// TwinCAT 3 PLC project Rohlik_Expansion
// ProgramVersion: 3.1.4024.0
// libraries:
//   CmpBitmapPool, * (System)
//   Tc2_EtherCAT, * (Beckhoff Automation GmbH)
//   Tc2_IoFunctions, * (Beckhoff Automation GmbH)
//   Tc2_MC2, * (Beckhoff Automation GmbH)
//   Tc2_ModbusSrv, * (Beckhoff Automation GmbH)
//   Tc2_Standard, * (Beckhoff Automation GmbH)
//   Tc2_SUPS, * (Beckhoff Automation GmbH)
//   Tc2_System, * (Beckhoff Automation GmbH)
//   Tc2_Utilities, * (Beckhoff Automation GmbH)
//   Tc3_Module, * (Beckhoff Automation GmbH)
//   Tc3_PackML_V2, * (Beckhoff Automation GmbH)
//   Util, * (System)
//   VisuDialogs, * (System)
// project tree:
//   02DUTs/ E_PMLUserUnitMode.TcDUT (not stored), E_UnitName.TcDUT (not stored), ModuleID.TcDUT (not stored), ST_ChangeIntoProduction.TcDUT (not stored), ST_UnitInfo.TcDUT (not stored)
//   Ads/ AbortToteRequestParams.TcDUT (not stored), AutostoreControlCommand.TcDUT (not stored), BarcodeValidationRequestParams.TcDUT (not stored), BarcodeVerificationResult.TcDUT (not stored), ButtonStatus.TcDUT (not stored), AirPressureStatus.TcDUT (not stored), DigitalInputStatus.TcDUT (not stored), DigitalOutputStatus.TcDUT (not stored), AutostoreStatus.TcDUT, EStopStatus.TcDUT (not stored), E_SAFETYDOOR.TcDUT (not stored), E_SafetyStates.TcDUT (not stored), FB_AirPressure_Subsystem.TcPOU, FB_HeartBeat_Subsystem.TcPOU, FB_Light_tower_module.TcPOU (not stored), FB_MachineControl_Subsystem.TcPOU (not stored), FB_Safety_Subsystem.TcPOU, FB_Tote_Subsystem.TcPOU, GeneralStatus.TcDUT (not stored), HeartbeatParams.TcDUT (not stored), InboundToteParams.TcDUT (not stored), InitToteRequestParams.TcDUT (not stored), LightCurtainStatus.TcDUT (not stored), MachineCommandStructure.TcDUT (not stored), MachineControlCommand.TcDUT (not stored), MachineControlCommand_1.TcDUT (not stored), MachineStatus.TcDUT (not stored), MethodCallReturnValue.TcDUT (not stored), ModelIdentifier.TcDUT (not stored), OrderToteCommand.TcDUT (not stored), OutboundToteParams.TcDUT (not stored), PerturbToteParams.TcDUT (not stored), SafetyDoorStatus.TcDUT (not stored), SafetyStatus.TcDUT (not stored), SensorStatus.TcDUT (not stored), StationMode.TcDUT (not stored), ST_BagOpen.TcDUT (not stored), ST_LightTower.TcDUT (not stored), SwapToteParams.TcDUT (not stored), ToteData.TcPOU (not stored), UpdateLightTowerParams.TcDUT (not stored), UpdateStationModeParams.TcDUT (not stored)
//   Ads/Ads/ BagOpeningStatus.TcPOU (not stored), ST_LightTowerAction.TcDUT (not stored)
//   GVLs/ GVL.TcGVL (not stored), GVL_SAFETY.TcGVL, G_HMI.TcGVL (not stored), G_IO.TcGVL (not stored), ST_Ifm_Qualifier.TcDUT (not stored), ST_Ifm_RX.TcDUT (not stored), ST_Ifm_TX.TcDUT (not stored), ST_IO_16.TcDUT (not stored), ST_SafetyIO.TcDUT (not stored)
//   / EtherCAT_Task.TcTTO (not stored), GlobalTextList.TcGTLO, MianTask.TcTTO (not stored), VisualizationManager.TcVMO (not stored), VISU_TASK.TcTTO (not stored)
//   LogTECH/ LogTechControlCmd.TcDUT (not stored), LogTechStatus.TcDUT (not stored), LogTechTransferStatus.TcDUT (not stored)
//   Mian/axis/ AxisHMI_Ex.TcVIS (not stored), E_HomingSteps.TcDUT (not stored), FB_MotionAxis_MC.TcPOU (not stored), MC_HomeAxis.TcPOU (not stored), ST_MotionAxis_MC.TcDUT (not stored)
//   Mian/DUTs/ BagStatus.TcDUT (not stored), Buffer_roller.TcDUT (not stored), E_Condition.TcDUT (not stored), E_LoadingStates.TcDUT (not stored), E_SampleStates.TcDUT (not stored), E_RollerStates.TcDUT (not stored), E_AutoStore_States.TcDUT (not stored), E_topic_sample.TcDUT (not stored), E_Transfer.TcDUT (not stored), E_WorkingStates.TcDUT, FB_DigitalInput.TcPOU (not stored), FB_GPWM.TcPOU (not stored), Inbound.TcDUT (not stored), I_Common.TcIO (not stored), OrderToteErrorStatus.TcDUT (not stored), Outbound.TcDUT (not stored), Prepare_Date_Time.TcPOU (not stored), Roller.TcDUT (not stored), Roller_x.TcDUT (not stored), Roller_y.TcDUT (not stored), ServerityLevelType.TcDUT (not stored), ST_Alarm_Hmi.TcDUT (not stored), ST_control_pannel.TcDUT (not stored), ST_EVENT.TcDUT (not stored), ST_safetyDoor.TcDUT (not stored), ToteStatus.TcDUT (not stored), ToteSubsystemWorkflowStatus.TcDUT (not stored), Valve.TcDUT (not stored)
//   Mian/ FB_Generic.TcPOU (not stored), FB_Machine.TcPOU (not stored), FB_mcp.TcPOU (not stored), FB_Sample.TcPOU (not stored), FB_loading_tote.TcPOU, FB_autoStore.TcPOU, FB_StateMachine.TcPOU, FB_working_tote.TcPOU, FB_Visu.TcPOU (not stored), FB_WriteLog.TcPOU (not stored), MAIN.TcPOU
//   PubSub/ E_Topics.TcDUT (not stored), I_PubSubService.TcIO (not stored), I_SubCallback.TcIO (not stored), KeyAndValue.TcDUT (not stored), PubSubData.TcDUT (not stored), PubSubService.TcPOU (not stored), ST_TracePublish.TcDUT (not stored), SubscriberCell.TcDUT (not stored)
//   VISUs/ ImagePool.TcIPO (not stored), visu_main.TcVIS (not stored)
//   VISUs/Templates/ visu_autoStore.TcVIS, VIS_TemplateCommand.TcVIS (not stored), VIS_TemplateKeys.TcVIS (not stored), VIS_TemplateMachine.TcVIS (not stored), VIS_TemplatePMLStateModel.TcVIS (not stored), VIS_TemplateToProduction.TcVIS (not stored), v_io_autoStore.TcVIS
//   VISUs/VISUs/ Menu.TcVIS, visu_2sys.TcVIS (not stored), visu_autoStore2.TcVIS, visu_loading.TcVIS (not stored), visu_operation.TcVIS, visu_sample.TcVIS (not stored), visu_manual.TcVIS, visu_working1.TcVIS (not stored), visu_autoStore1.TcVIS (not stored), visu_working2.TcVIS (not stored), v_alarm.TcVIS (not stored), v_io_loading.TcVIS (not stored), v_io_working1.TcVIS (not stored), v_io_working2.TcVIS
// real-time tasks:
//   TASK PlcTask: cycle T#4ms, priority 20, ADS port 350
//   TASK EtherCAT_Task: cycle T#2ms, priority 2, ADS port 351
//   TASK VISU_TASK: cycle T#100000us, priority 30, ADS port 352
// motion (NC):
//   TASK NC-Task 1 SAF: cycle T#2ms, priority 4, ADS port 501
//   TASK NC-Task 1 SVB: cycle T#10ms, priority 8, ADS port 511
//   AXIS lift_motor (id 3)
//     Velo: SlowManual=5, FastManual=20
//     PositionAreaControl: Enable=false
//     OtherSettings: AllowMotionCmdToSlave=true
//     encoder EncType=19
//       EncPara: ScaleFactorNumerator=3.333333333333, ScaleFactorDenominator=8388608, Inverse=true, MaxCount=#xffffffff, ReferenceSystem=1
//         SoftEndMinControl: Enable=true, Range=-5
//         SoftEndMaxControl: Enable=true, Range=800
//         Inc: RefSoftSyncMask=#x00800000
//     drive DrvType=16
//       DrvPara: Inverse=true, MaxCount=#xffffffff, DriveControlDWord=#x00020100
//         Analog: TorqueSetpointScale=10, ScaleFactorActTorque=0.1
//         TimeComp: TaskDelayCycles=1
//     controller CtrType=1
//       CtrPara: PriorControlFactor=1
//         PosDiffControl: Enable=false
//         Observer: BandWidth=20
//   AXIS working1_lift_motor (id 4)
//     PositionAreaControl: Enable=false
//     OtherSettings: AllowMotionCmdToSlave=true
//     encoder EncType=19
//       EncPara: ScaleFactorNumerator=5, ScaleFactorDenominator=8388608, Inverse=true, MaxCount=#xffffffff, ReferenceSystem=1
//         SoftEndMinControl: Enable=true, Range=-5
//         SoftEndMaxControl: Enable=true, Range=140
//         Inc: RefSoftSyncMask=#x00800000
//     drive DrvType=16
//       DrvPara: Inverse=true, MaxCount=#xffffffff, DriveControlDWord=#x00020100
//         Analog: TorqueSetpointScale=10, ScaleFactorActTorque=0.1
//         TimeComp: TaskDelayCycles=1
//     controller CtrType=1
//       CtrPara: PriorControlFactor=1
//         PosDiffControl: Enable=false
//         Observer: BandWidth=20
//   AXIS working1_open_bag (id 5)
//     General: UnitName=°
//     Dynamic: Acceleration=75, Deceleration=75, Jerk=112.5
//     Velo: SlowManual=1, FastManual=5, Maximum=300
//     PositionAreaControl: Enable=false
//     OtherSettings: AllowMotionCmdToSlave=true
//     encoder EncType=19
//       EncPara: ScaleFactorNumerator=36, ScaleFactorDenominator=8388608, MaxCount=#xffffffff, ReferenceSystem=1
//         SoftEndMinControl: Enable=true
//         SoftEndMaxControl: Enable=true, Range=60
//         Inc: RefSoftSyncMask=#x00800000
//     drive DrvType=16
//       DrvPara: MaxCount=#xffffffff, DriveControlDWord=#x00020100
//         Analog: TorqueSetpointScale=10, ScaleFactorActTorque=0.1
//         TimeComp: TaskDelayCycles=1
//     controller CtrType=1
//       CtrPara: PriorControlFactor=1
//         PosDiffControl: Enable=false
//         Observer: BandWidth=20
//   AXIS working2_lift_motor (id 1)
//     PositionAreaControl: Enable=false
//     OtherSettings: AllowMotionCmdToSlave=true
//     encoder EncType=19
//       EncPara: ScaleFactorNumerator=5, ScaleFactorDenominator=8388608, Inverse=true, MaxCount=#xffffffff, ReferenceSystem=1
//         SoftEndMinControl: Enable=true, Range=-5
//         SoftEndMaxControl: Enable=true, Range=140
//         Inc: RefSoftSyncMask=#x00800000
//     drive DrvType=16
//       DrvPara: Inverse=true, MaxCount=#xffffffff, DriveControlDWord=#x00020100
//         Analog: TorqueSetpointScale=10, ScaleFactorActTorque=0.1
//         TimeComp: TaskDelayCycles=1
//     controller CtrType=1
//       CtrPara: PriorControlFactor=1
//         PosDiffControl: Enable=false
//         Observer: BandWidth=20
//   AXIS working2_open_bag (id 2)
//     General: UnitName=°
//     Dynamic: Acceleration=75, Deceleration=75, Jerk=112.5
//     Velo: Maximum=300
//     PositionAreaControl: Enable=false
//     OtherSettings: AllowMotionCmdToSlave=true
//     encoder EncType=19
//       EncPara: ScaleFactorNumerator=36, ScaleFactorDenominator=8388608, MaxCount=#xffffffff, ReferenceSystem=1
//         SoftEndMinControl: Enable=true
//         SoftEndMaxControl: Enable=true, Range=60
//         Inc: RefSoftSyncMask=#x00800000
//     drive DrvType=16
//       DrvPara: MaxCount=#xffffffff, DriveControlDWord=#x00020100
//         Analog: TorqueSetpointScale=10, ScaleFactorActTorque=0.1
//         TimeComp: TaskDelayCycles=1
//     controller CtrType=1
//       CtrPara: PriorControlFactor=1
//         PosDiffControl: Enable=false
//         Observer: BandWidth=20
//   AXIS autostore1_transfer (id 12)
//     General: UnitName=°
//     Dynamic: Acceleration=75, Deceleration=75, Jerk=112.5
//     Velo: Maximum=600
//     PositionAreaControl: Enable=false
//     OtherSettings: AllowMotionCmdToSlave=true
//     encoder EncType=19
//       EncPara: ScaleFactorNumerator=34.6, ScaleFactorDenominator=8388608, Inverse=true, MaxCount=#xffffffff, ReferenceSystem=1
//         SoftEndMaxControl: Range=56
//         Inc: RefSoftSyncMask=#x00800000
//     drive DrvType=16
//       DrvPara: Inverse=true, MaxCount=#xffffffff, DriveControlDWord=#x00000100
//         Analog: TorqueSetpointScale=10, ScaleFactorActTorque=0.1
//         TimeComp: TaskDelayCycles=1
//     controller CtrType=1
//       CtrPara: PriorControlFactor=1
//         PosDiffControl: Enable=false
//         Observer: BandWidth=20
//   AXIS autostore1_lift (id 13)
//     General: UnitName=°
//     Dynamic: Acceleration=75, Deceleration=75, Jerk=112.5
//     Velo: Maximum=400
//     PositionAreaControl: Enable=false
//     OtherSettings: AllowMotionCmdToSlave=true
//     encoder EncType=19
//       EncPara: ScaleFactorNumerator=40, ScaleFactorDenominator=8388608, MaxCount=#xffffffff, ReferenceSystem=1
//         SoftEndMaxControl: Range=56
//         Inc: RefSoftSyncMask=#x00800000
//     drive DrvType=16
//       DrvPara: MaxCount=#xffffffff, DriveControlDWord=#x00000100
//         Analog: TorqueSetpointScale=10, ScaleFactorActTorque=0.1
//         TimeComp: TaskDelayCycles=1
//     controller CtrType=1
//       CtrPara: PriorControlFactor=1
//         PosDiffControl: Enable=false
//         Observer: BandWidth=20
//   AXIS autostore2_lift (id 7)
//     General: UnitName=°
//     Dynamic: Acceleration=75, Deceleration=75, Jerk=112.5
//     Velo: Maximum=400
//     PositionAreaControl: Enable=false
//     OtherSettings: AllowMotionCmdToSlave=true
//     encoder EncType=19
//       EncPara: ScaleFactorNumerator=40, ScaleFactorDenominator=8388608, MaxCount=#xffffffff, ReferenceSystem=1
//         SoftEndMaxControl: Range=56
//         Inc: RefSoftSyncMask=#x00800000
//     drive DrvType=16
//       DrvPara: MaxCount=#xffffffff, DriveControlDWord=#x00020100
//         Analog: TorqueSetpointScale=10, ScaleFactorActTorque=0.1
//         TimeComp: TaskDelayCycles=1
//     controller CtrType=1
//       CtrPara: PriorControlFactor=1
//         PosDiffControl: Enable=false
//         Observer: BandWidth=20
//   AXIS autostore2_transfer (id 6)
//     General: UnitName=°
//     Dynamic: Acceleration=75, Deceleration=75, Jerk=112.5
//     Velo: Maximum=600
//     PositionAreaControl: Enable=false
//     OtherSettings: AllowMotionCmdToSlave=true
//     encoder EncType=19
//       EncPara: ScaleFactorNumerator=34.6, ScaleFactorDenominator=8388608, Inverse=true, MaxCount=#xffffffff, ReferenceSystem=1
//         SoftEndMaxControl: Range=56
//         Inc: RefSoftSyncMask=#x00800000
//     drive DrvType=16
//       DrvPara: Inverse=true, MaxCount=#xffffffff, DriveControlDWord=#x00020100
//         Analog: TorqueSetpointScale=10, ScaleFactorActTorque=0.1
//         TimeComp: TaskDelayCycles=1
//     controller CtrType=1
//       CtrPara: PriorControlFactor=1
//         PosDiffControl: Enable=false
//         Observer: BandWidth=20
// I/O:
//   DEVICE Device 2 (RT-Ethernet Adapter)
//   DEVICE MCP, AmsNetId 192.168.17.27.4.1
//     Box 1 (CU2508) [CU2508 Ethernet Port]
//     MCP-EK1100 [EK1100 EtherCAT Coupler (2A E-Bus)]
//       DI0 [EL1809 16Ch. Dig. Input 24V, 3ms]
//       DI1 [EL1809 16Ch. Dig. Input 24V, 3ms]
//       DO0 [EL2809 16Ch. Dig. Output 24V, 0.5A]
//       DO1 [EL2809 16Ch. Dig. Output 24V, 0.5A]
//       Term 7 (EL6910) [EL6910, TwinSAFE PLC]
//       SI0 [EL1904, 4 Ch. Safety Input 24V, TwinSAFE]
//         modules: Module 1 (FSOES)
//       SI1 [EL1904, 4 Ch. Safety Input 24V, TwinSAFE]
//         modules: Module 1 (FSOES)
//       SI2 [EL1904, 4 Ch. Safety Input 24V, TwinSAFE]
//         modules: Module 1 (FSOES)
//       SI3 [EL1904, 4 Ch. Safety Input 24V, TwinSAFE]
//         modules: Module 1 (FSOES)
//       SO0 [EL2904, 4 Ch. Safety Output 24V, 0.5A, TwinSAFE]
//         modules: Module 1 (FSOES), Module 2 (DO)
//       SO4 [EL2904, 4 Ch. Safety Output 24V, 0.5A, TwinSAFE]
//         modules: Module 1 (FSOES), Module 2 (DO)
//       Term 50 (EL9410) [EL9410 E-Bus Power Supplier  (Diagnostics)]
//       Term 13 (EL3064) [EL3064 4Ch. Ana. Input 0-10V]
//       SI7 [EL1904, 4 Ch. Safety Input 24V, TwinSAFE]
//         modules: Module 1 (FSOES)
//       SI8 [EL1904, 4 Ch. Safety Input 24V, TwinSAFE]
//         modules: Module 1 (FSOES)
//       SO5 [EL2904, 4 Ch. Safety Output 24V, 0.5A, TwinSAFE]
//         modules: Module 1 (FSOES), Module 2 (DO)
//       SO6 [EL2904, 4 Ch. Safety Output 24V, 0.5A, TwinSAFE]
//         modules: Module 1 (FSOES), Module 2 (DO)
//       Term 14 (EL6631-0010) [EL6631-0010 PROFINET IO Device]
//       Term 15 (EL9011) [EL9011 End Terminal]
//   DEVICE Lift, AmsNetId 192.168.17.27.5.1
//     Box 16 (CU2508) [CU2508 Ethernet Port]
//     Term 17 (EK1100) [EK1100 EtherCAT Coupler (2A E-Bus)]
//       DI2 [EL1809 16Ch. Dig. Input 24V, 3ms]
//       DI3 [EL1809 16Ch. Dig. Input 24V, 3ms]
//       DO2 [EL2809 16Ch. Dig. Output 24V, 0.5A]
//       DO3 [EL2809 16Ch. Dig. Output 24V, 0.5A]
//       SI4 [EL1904, 4 Ch. Safety Input 24V, TwinSAFE]
//         modules: Module 1 (FSOES)
//       SI5 [EL1904, 4 Ch. Safety Input 24V, TwinSAFE]
//         modules: Module 1 (FSOES)
//       SI6 [EL1904, 4 Ch. Safety Input 24V, TwinSAFE]
//         modules: Module 1 (FSOES)
//       SO1 [EL2904, 4 Ch. Safety Output 24V, 0.5A, TwinSAFE]
//         modules: Module 1 (FSOES), Module 2 (DO)
//       Term 10 (EL9011) [EL9011 End Terminal]
//     lift_lift [SV660_1Axis_00915]
//     Box 26 (ifm IO-Link Master AL1332) [ifm IO-Link Master AL1332]
//       modules: Module 1 (IOL_4/4_I/O-Bytes), Module 2 (IOL_4/4_I/O-Bytes), Module 3 (IOL_4/4_I/O-Bytes), Module 4 (IOL_4/4_I/O-Bytes), Module 5 (IOL_4/4_I/O-Bytes), Module 6 (IOL_4/4_I/O-Bytes), Module 7 (IOL_4/4_I/O-Bytes), Module 8 (IOL_4/4_I/O-Bytes)
//   DEVICE Place1, AmsNetId 192.168.17.27.6.1
//     Box 26 (CU2508) [CU2508 Ethernet Port]
//     Term 27 (EK1100) [EK1100 EtherCAT Coupler (2A E-Bus)]
//       DI4 [EL1809 16Ch. Dig. Input 24V, 3ms]
//       DI5 [EL1809 16Ch. Dig. Input 24V, 3ms]
//       DO4 [EL2809 16Ch. Dig. Output 24V, 0.5A]
//       SO2 [EL2904, 4 Ch. Safety Output 24V, 0.5A, TwinSAFE]
//         modules: Module 1 (FSOES), Module 2 (DO)
//       Term 53 (EL9410) [EL9410 E-Bus Power Supplier  (Diagnostics)]
//       DO6 [EL2809 16Ch. Dig. Output 24V, 0.5A]
//       Term 9 (EL9011) [EL9011 End Terminal]
//     place1_lift [SV660_1Axis_00915]
//     place_openbag [SV660_1Axis_00915]
//     Box 36 (ifm IO-Link Master AL1332) [ifm IO-Link Master AL1332]
//       modules: Module 1 (IOL_4/4_I/O-Bytes), Module 2 (IOL_4/4_I/O-Bytes), Module 3 (IOL_4/4_I/O-Bytes), Module 4 (IOL_4/4_I/O-Bytes), Module 5 (IOL_4/4_I/O-Bytes), Module 6 (IOL_4/4_I/O-Bytes), Module 7 (IOL_4/4_I/O-Bytes), Module 8 (IOL_4/4_I/O-Bytes)
//   DEVICE Place2, AmsNetId 192.168.17.27.7.1
//     Box 35 (CU2508) [CU2508 Ethernet Port]
//     Term 36 (EK1100) [EK1100 EtherCAT Coupler (2A E-Bus)]
//       DI6 [EL1809 16Ch. Dig. Input 24V, 3ms]
//       DI7 [EL1809 16Ch. Dig. Input 24V, 3ms]
//       DO5 [EL2809 16Ch. Dig. Output 24V, 0.5A]
//       SO3 [EL2904, 4 Ch. Safety Output 24V, 0.5A, TwinSAFE]
//         modules: Module 1 (FSOES), Module 2 (DO)
//       Term 51 (EL9410) [EL9410 E-Bus Power Supplier  (Diagnostics)]
//       DO7 [EL2809 16Ch. Dig. Output 24V, 0.5A]
//       Term 9 (EL9011) [EL9011 End Terminal]
//     place2_lift [SV660_1Axis_00915]
//     place2_openbag [SV660_1Axis_00915]
//     Box 46 (ifm IO-Link Master AL1332) [ifm IO-Link Master AL1332]
//       modules: Module 1 (IOL_4/4_I/O-Bytes), Module 2 (IOL_4/4_I/O-Bytes), Module 3 (IOL_4/4_I/O-Bytes), Module 4 (IOL_4/4_I/O-Bytes), Module 5 (IOL_4/4_I/O-Bytes), Module 6 (IOL_4/4_I/O-Bytes), Module 7 (IOL_4/4_I/O-Bytes), Module 8 (IOL_4/4_I/O-Bytes)
//   DEVICE Device 1 (EtherCAT Automation Protocol), AmsNetId 192.168.11.159.2.1
//   DEVICE autoStore1, AmsNetId 192.168.11.159.8.1
//     Box 55 (CU2508) [CU2508 Ethernet Port]
//     Term 56 (EK1100) [EK1100 EtherCAT Coupler (2A E-Bus)]
//       DI20 [EL1809 16Ch. Dig. Input 24V, 3ms]
//       Term 6 (EL9011) [EL9011 End Terminal]
//     autostore1_transfer [SV660_1Axis_00916]
//     autostore1_lift [SV660_1Axis_00916]
//   DEVICE autoStore2, AmsNetId 192.168.11.159.10.1
//     Box 65 (CU2508) [CU2508 Ethernet Port]
//     Term 70 (EK1100) [EK1100 EtherCAT Coupler (2A E-Bus)]
//       DI21 [EL1809 16Ch. Dig. Input 24V, 3ms]
//       Term 10 (EL9011) [EL9011 End Terminal]
//     autostore2_transfer [SV660_1Axis_00916]
//     autostore2_lift [SV660_1Axis_00916]
// variable links:
//   Lift <-> MCP/MCP-EK1100/Term 7 (EL6910)
//     Term 17 (EK1100)/SI5/Module 1 (FSOES)/RxPDO/FSOE <-> ConnectionInputs/Message_29 TxPDO
//     Term 17 (EK1100)/SI6/Module 1 (FSOES)/RxPDO/FSOE <-> ConnectionInputs/Message_30 TxPDO
//     Term 17 (EK1100)/SO1/Module 1 (FSOES)/TxPDO/FSOE <-> ConnectionOutputs/Message_31 RxPDO
//   MCP <-> Lift/Term 17 (EK1100)/SI4
//     MCP-EK1100/Term 7 (EL6910)/ConnectionInputs/Message_28 TxPDO <-> Module 1 (FSOES)/RxPDO/FSOE
//     MCP-EK1100/Term 7 (EL6910)/ConnectionOutputs/Message_28 RxPDO <-> Module 1 (FSOES)/TxPDO/FSOE
//   MCP <-> Lift/Term 17 (EK1100)/SI5
//     MCP-EK1100/Term 7 (EL6910)/ConnectionOutputs/Message_29 RxPDO <-> Module 1 (FSOES)/TxPDO/FSOE
//   MCP <-> Lift/Term 17 (EK1100)/SI6
//     MCP-EK1100/Term 7 (EL6910)/ConnectionOutputs/Message_30 RxPDO <-> Module 1 (FSOES)/TxPDO/FSOE
//   MCP <-> Lift/Term 17 (EK1100)/SO1
//     MCP-EK1100/Term 7 (EL6910)/ConnectionInputs/Message_31 TxPDO <-> Module 1 (FSOES)/RxPDO/FSOE
//   MCP <-> MCP/MCP-EK1100/SI0
//     MCP-EK1100/Term 7 (EL6910)/ConnectionInputs/Message_22 TxPDO <-> Module 1 (FSOES)/RxPDO/FSOE
//     MCP-EK1100/Term 7 (EL6910)/ConnectionOutputs/Message_22 RxPDO <-> Module 1 (FSOES)/TxPDO/FSOE
//   MCP <-> MCP/MCP-EK1100/SI1
//     MCP-EK1100/Term 7 (EL6910)/ConnectionInputs/Message_23 TxPDO <-> Module 1 (FSOES)/RxPDO/FSOE
//   MCP <-> MCP/MCP-EK1100/SI2
//     MCP-EK1100/Term 7 (EL6910)/ConnectionOutputs/Message_24 RxPDO <-> Module 1 (FSOES)/TxPDO/FSOE
//   MCP <-> MCP/MCP-EK1100/SI3
//     MCP-EK1100/Term 7 (EL6910)/ConnectionInputs/Message_27 TxPDO <-> Module 1 (FSOES)/RxPDO/FSOE
//   MCP <-> MCP/MCP-EK1100/SO0
//     MCP-EK1100/Term 7 (EL6910)/ConnectionInputs/Message_26 TxPDO <-> Module 1 (FSOES)/RxPDO/FSOE
//   MCP <-> MCP/MCP-EK1100/SO5
//     MCP-EK1100/Term 7 (EL6910)/ConnectionOutputs/Message_71 RxPDO <-> Module 1 (FSOES)/TxPDO/FSOE
//   MCP <-> MCP/MCP-EK1100/SO6
//     MCP-EK1100/Term 7 (EL6910)/ConnectionInputs/Message_72 TxPDO <-> Module 1 (FSOES)/RxPDO/FSOE
//   MCP <-> MCP/MCP-EK1100/Term 7 (EL6910)
//     MCP-EK1100/SI1/Module 1 (FSOES)/TxPDO/FSOE <-> ConnectionOutputs/Message_23 RxPDO
//     MCP-EK1100/SI3/Module 1 (FSOES)/TxPDO/FSOE <-> ConnectionOutputs/Message_27 RxPDO
//     MCP-EK1100/SI2/Module 1 (FSOES)/RxPDO/FSOE <-> ConnectionInputs/Message_24 TxPDO
//     MCP-EK1100/SO0/Module 1 (FSOES)/TxPDO/FSOE <-> ConnectionOutputs/Message_26 RxPDO
//     MCP-EK1100/SO4/Module 1 (FSOES)/TxPDO/FSOE <-> ConnectionOutputs/Message_36 RxPDO
//     MCP-EK1100/SO6/Module 1 (FSOES)/TxPDO/FSOE <-> ConnectionOutputs/Message_72 RxPDO
//     MCP-EK1100/SO4/Module 1 (FSOES)/RxPDO/FSOE <-> ConnectionInputs/Message_36 TxPDO
//     MCP-EK1100/SO5/Module 1 (FSOES)/RxPDO/FSOE <-> ConnectionInputs/Message_71 TxPDO
//   MCP <-> Place2/Term 36 (EK1100)/SO3
//     MCP-EK1100/Term 7 (EL6910)/ConnectionInputs/Message_33 TxPDO <-> Module 1 (FSOES)/RxPDO/FSOE
//     MCP-EK1100/Term 7 (EL6910)/ConnectionOutputs/Message_33 RxPDO <-> Module 1 (FSOES)/TxPDO/FSOE
//   Place1 <-> MCP/MCP-EK1100/Term 7 (EL6910)
//     Term 27 (EK1100)/SO2/Module 1 (FSOES)/RxPDO/FSOE <-> ConnectionInputs/Message_32 TxPDO
//     Term 27 (EK1100)/SO2/Module 1 (FSOES)/TxPDO/FSOE <-> ConnectionOutputs/Message_32 RxPDO
//   NC-Task 1 SAF/Axes/autostore1_lift <-> autoStore1/autostore1_lift
//     Drive/Inputs/In/nDataIn1 <-> Inputs/Following error actual value
//     Drive/Inputs/In/nDataIn3[0] <-> Inputs/Torque actual value
//     Drive/Inputs/In/nDcOutputTime <-> InfoData/DcOutputShift
//     Drive/Inputs/In/nState1 <-> Inputs/Statusword
//     Drive/Inputs/In/nState2 <-> Inputs/Statusword @bit 8
//     Drive/Inputs/In/nState4 @bit 1 <-> WcState/InputToggle
//     Drive/Inputs/In/nState4 <-> WcState/WcState
//     Drive/Outputs/Out/nCtrl1 <-> Outputs/Controlword
//     Drive/Outputs/Out/nCtrl2 <-> Outputs/Controlword @bit 8
//     Drive/Outputs/Out/nDataOut1 <-> Outputs/Target position
//     Enc/Inputs/In/nDataIn1 <-> Inputs/Position actual value
//     Enc/Inputs/In/nDataIn3 <-> Inputs/Touch probe pos1 pos value
//     Enc/Inputs/In/nDataIn5 <-> Inputs/Touch probe pos2 pos value
//     Enc/Inputs/In/nDcInputTime <-> InfoData/DcInputShift
//     Enc/Inputs/In/nState4 @bit 1 <-> WcState/InputToggle
//     Enc/Inputs/In/nState4 <-> WcState/WcState
//     Enc/Inputs/In/nState5 <-> Inputs/Touch probe status
//     Enc/Inputs/In/nState6 <-> Inputs/Touch probe status @bit 8
//     Enc/Outputs/Out/nCtrl5 <-> Outputs/Touch probe function
//     Enc/Outputs/Out/nCtrl6 <-> Outputs/Touch probe function @bit 8
//   NC-Task 1 SAF/Axes/autostore1_transfer <-> autoStore1/autostore1_transfer
//     Drive/Inputs/In/nDataIn1 <-> Inputs/Following error actual value
//     Drive/Inputs/In/nDataIn3[0] <-> Inputs/Torque actual value
//     Drive/Inputs/In/nDcOutputTime <-> InfoData/DcOutputShift
//     Drive/Inputs/In/nState1 <-> Inputs/Statusword
//     Drive/Inputs/In/nState2 <-> Inputs/Statusword @bit 8
//     Drive/Inputs/In/nState4 @bit 1 <-> WcState/InputToggle
//     Drive/Inputs/In/nState4 <-> WcState/WcState
//     Drive/Outputs/Out/nCtrl1 <-> Outputs/Controlword
//     Drive/Outputs/Out/nCtrl2 <-> Outputs/Controlword @bit 8
//     Drive/Outputs/Out/nDataOut1 <-> Outputs/Target position
//     Enc/Inputs/In/nDataIn1 <-> Inputs/Position actual value
//     Enc/Inputs/In/nDataIn3 <-> Inputs/Touch probe pos1 pos value
//     Enc/Inputs/In/nDataIn5 <-> Inputs/Touch probe pos2 pos value
//     Enc/Inputs/In/nDcInputTime <-> InfoData/DcInputShift
//     Enc/Inputs/In/nState4 @bit 1 <-> WcState/InputToggle
//     Enc/Inputs/In/nState4 <-> WcState/WcState
//     Enc/Inputs/In/nState5 <-> Inputs/Touch probe status
//     Enc/Inputs/In/nState6 <-> Inputs/Touch probe status @bit 8
//     Enc/Outputs/Out/nCtrl5 <-> Outputs/Touch probe function
//     Enc/Outputs/Out/nCtrl6 <-> Outputs/Touch probe function @bit 8
//   NC-Task 1 SAF/Axes/autostore2_lift <-> autoStore2/autostore2_lift
//     Drive/Inputs/In/nDataIn1 <-> Inputs/Following error actual value
//     Drive/Inputs/In/nDataIn3[0] <-> Inputs/Torque actual value
//     Drive/Inputs/In/nDcOutputTime <-> InfoData/DcOutputShift
//     Drive/Inputs/In/nState1 <-> Inputs/Statusword
//     Drive/Inputs/In/nState2 <-> Inputs/Statusword @bit 8
//     Drive/Inputs/In/nState4 @bit 1 <-> WcState/InputToggle
//     Drive/Inputs/In/nState4 <-> WcState/WcState
//     Drive/Outputs/Out/nCtrl1 <-> Outputs/Controlword
//     Drive/Outputs/Out/nCtrl2 <-> Outputs/Controlword @bit 8
//     Drive/Outputs/Out/nDataOut1 <-> Outputs/Target position
//     Enc/Inputs/In/nDataIn1 <-> Inputs/Position actual value
//     Enc/Inputs/In/nDataIn3 <-> Inputs/Touch probe pos1 pos value
//     Enc/Inputs/In/nDataIn5 <-> Inputs/Touch probe pos2 pos value
//     Enc/Inputs/In/nDcInputTime <-> InfoData/DcInputShift
//     Enc/Inputs/In/nState4 @bit 1 <-> WcState/InputToggle
//     Enc/Inputs/In/nState4 <-> WcState/WcState
//     Enc/Inputs/In/nState5 <-> Inputs/Touch probe status
//     Enc/Inputs/In/nState6 <-> Inputs/Touch probe status @bit 8
//     Enc/Outputs/Out/nCtrl5 <-> Outputs/Touch probe function
//     Enc/Outputs/Out/nCtrl6 <-> Outputs/Touch probe function @bit 8
//   NC-Task 1 SAF/Axes/autostore2_transfer <-> autoStore2/autostore2_transfer
//     Drive/Inputs/In/nDataIn1 <-> Inputs/Following error actual value
//     Drive/Inputs/In/nDataIn3[0] <-> Inputs/Torque actual value
//     Drive/Inputs/In/nDcOutputTime <-> InfoData/DcOutputShift
//     Drive/Inputs/In/nState1 <-> Inputs/Statusword
//     Drive/Inputs/In/nState2 <-> Inputs/Statusword @bit 8
//     Drive/Inputs/In/nState4 @bit 1 <-> WcState/InputToggle
//     Drive/Inputs/In/nState4 <-> WcState/WcState
//     Drive/Outputs/Out/nCtrl1 <-> Outputs/Controlword
//     Drive/Outputs/Out/nCtrl2 <-> Outputs/Controlword @bit 8
//     Drive/Outputs/Out/nDataOut1 <-> Outputs/Target position
//     Enc/Inputs/In/nDataIn1 <-> Inputs/Position actual value
//     Enc/Inputs/In/nDataIn3 <-> Inputs/Touch probe pos1 pos value
//     Enc/Inputs/In/nDataIn5 <-> Inputs/Touch probe pos2 pos value
//     Enc/Inputs/In/nDcInputTime <-> InfoData/DcInputShift
//     Enc/Inputs/In/nState4 @bit 1 <-> WcState/InputToggle
//     Enc/Inputs/In/nState4 <-> WcState/WcState
//     Enc/Inputs/In/nState5 <-> Inputs/Touch probe status
//     Enc/Inputs/In/nState6 <-> Inputs/Touch probe status @bit 8
//     Enc/Outputs/Out/nCtrl5 <-> Outputs/Touch probe function
//     Enc/Outputs/Out/nCtrl6 <-> Outputs/Touch probe function @bit 8
//   NC-Task 1 SAF/Axes/lift_motor <-> Lift/lift_lift
//     Drive/Inputs/In/nDataIn1 <-> Inputs/Following error actual value
//     Drive/Inputs/In/nDataIn3[0] <-> Inputs/Torque actual value
//     Drive/Inputs/In/nDcOutputTime <-> InfoData/DcOutputShift
//     Drive/Inputs/In/nState1 <-> Inputs/Statusword
//     Drive/Inputs/In/nState2 <-> Inputs/Statusword @bit 8
//     Drive/Inputs/In/nState4 @bit 1 <-> WcState/InputToggle
//     Drive/Inputs/In/nState4 <-> WcState/WcState
//     Drive/Outputs/Out/nCtrl1 <-> Outputs/Controlword
//     Drive/Outputs/Out/nCtrl2 <-> Outputs/Controlword @bit 8
//     Drive/Outputs/Out/nDataOut1 <-> Outputs/Target position
//     Enc/Inputs/In/nDataIn1 <-> Inputs/Position actual value
//     Enc/Inputs/In/nDataIn3 <-> Inputs/Touch probe pos1 pos value
//     Enc/Inputs/In/nDataIn5 <-> Inputs/Touch probe pos2 pos value
//     Enc/Inputs/In/nDcInputTime <-> InfoData/DcInputShift
//     Enc/Inputs/In/nState4 @bit 1 <-> WcState/InputToggle
//     Enc/Inputs/In/nState4 <-> WcState/WcState
//     Enc/Inputs/In/nState5 <-> Inputs/Touch probe status
//     Enc/Inputs/In/nState6 <-> Inputs/Touch probe status @bit 8
//     Enc/Outputs/Out/nCtrl5 <-> Outputs/Touch probe function
//     Enc/Outputs/Out/nCtrl6 <-> Outputs/Touch probe function @bit 8
//   NC-Task 1 SAF/Axes/working1_lift_motor <-> Place1/place1_lift
//     Drive/Inputs/In/nDataIn1 <-> Inputs/Following error actual value
//     Drive/Inputs/In/nDataIn3[0] <-> Inputs/Torque actual value
//     Drive/Inputs/In/nDcOutputTime <-> InfoData/DcOutputShift
//     Drive/Inputs/In/nState1 <-> Inputs/Statusword
//     Drive/Inputs/In/nState2 <-> Inputs/Statusword @bit 8
//     Drive/Inputs/In/nState4 @bit 1 <-> WcState/InputToggle
//     Drive/Inputs/In/nState4 <-> WcState/WcState
//     Drive/Outputs/Out/nCtrl1 <-> Outputs/Controlword
//     Drive/Outputs/Out/nCtrl2 <-> Outputs/Controlword @bit 8
//     Drive/Outputs/Out/nDataOut1 <-> Outputs/Target position
//     Enc/Inputs/In/nDataIn1 <-> Inputs/Position actual value
//     Enc/Inputs/In/nDataIn3 <-> Inputs/Touch probe pos1 pos value
//     Enc/Inputs/In/nDataIn5 <-> Inputs/Touch probe pos2 pos value
//     Enc/Inputs/In/nDcInputTime <-> InfoData/DcInputShift
//     Enc/Inputs/In/nState4 @bit 1 <-> WcState/InputToggle
//     Enc/Inputs/In/nState4 <-> WcState/WcState
//     Enc/Inputs/In/nState5 <-> Inputs/Touch probe status
//     Enc/Inputs/In/nState6 <-> Inputs/Touch probe status @bit 8
//     Enc/Outputs/Out/nCtrl5 <-> Outputs/Touch probe function
//     Enc/Outputs/Out/nCtrl6 <-> Outputs/Touch probe function @bit 8
//   NC-Task 1 SAF/Axes/working1_open_bag <-> Place1/place_openbag
//     Drive/Inputs/In/nDataIn1 <-> Inputs/Following error actual value
//     Drive/Inputs/In/nDataIn3[0] <-> Inputs/Torque actual value
//     Drive/Inputs/In/nDcOutputTime <-> InfoData/DcOutputShift
//     Drive/Inputs/In/nState1 <-> Inputs/Statusword
//     Drive/Inputs/In/nState2 <-> Inputs/Statusword @bit 8
//     Drive/Inputs/In/nState4 @bit 1 <-> WcState/InputToggle
//     Drive/Inputs/In/nState4 <-> WcState/WcState
//     Drive/Outputs/Out/nCtrl1 <-> Outputs/Controlword
//     Drive/Outputs/Out/nCtrl2 <-> Outputs/Controlword @bit 8
//     Drive/Outputs/Out/nDataOut1 <-> Outputs/Target position
//     Enc/Inputs/In/nDataIn1 <-> Inputs/Position actual value
//     Enc/Inputs/In/nDataIn3 <-> Inputs/Touch probe pos1 pos value
//     Enc/Inputs/In/nDataIn5 <-> Inputs/Touch probe pos2 pos value
//     Enc/Inputs/In/nDcInputTime <-> InfoData/DcInputShift
//     Enc/Inputs/In/nState4 @bit 1 <-> WcState/InputToggle
//     Enc/Inputs/In/nState4 <-> WcState/WcState
//     Enc/Inputs/In/nState5 <-> Inputs/Touch probe status
//     Enc/Inputs/In/nState6 <-> Inputs/Touch probe status @bit 8
//     Enc/Outputs/Out/nCtrl5 <-> Outputs/Touch probe function
//     Enc/Outputs/Out/nCtrl6 <-> Outputs/Touch probe function @bit 8
//   NC-Task 1 SAF/Axes/working2_lift_motor <-> Place2/place2_lift
//     Drive/Inputs/In/nDataIn1 <-> Inputs/Following error actual value
//     Drive/Inputs/In/nDataIn3[0] <-> Inputs/Torque actual value
//     Drive/Inputs/In/nDcOutputTime <-> InfoData/DcOutputShift
//     Drive/Inputs/In/nState1 <-> Inputs/Statusword
//     Drive/Inputs/In/nState2 <-> Inputs/Statusword @bit 8
//     Drive/Inputs/In/nState4 @bit 1 <-> WcState/InputToggle
//     Drive/Inputs/In/nState4 <-> WcState/WcState
//     Drive/Outputs/Out/nCtrl1 <-> Outputs/Controlword
//     Drive/Outputs/Out/nCtrl2 <-> Outputs/Controlword @bit 8
//     Drive/Outputs/Out/nDataOut1 <-> Outputs/Target position
//     Enc/Inputs/In/nDataIn1 <-> Inputs/Position actual value
//     Enc/Inputs/In/nDataIn3 <-> Inputs/Touch probe pos1 pos value
//     Enc/Inputs/In/nDataIn5 <-> Inputs/Touch probe pos2 pos value
//     Enc/Inputs/In/nDcInputTime <-> InfoData/DcInputShift
//     Enc/Inputs/In/nState4 @bit 1 <-> WcState/InputToggle
//     Enc/Inputs/In/nState4 <-> WcState/WcState
//     Enc/Inputs/In/nState5 <-> Inputs/Touch probe status
//     Enc/Inputs/In/nState6 <-> Inputs/Touch probe status @bit 8
//     Enc/Outputs/Out/nCtrl5 <-> Outputs/Touch probe function
//     Enc/Outputs/Out/nCtrl6 <-> Outputs/Touch probe function @bit 8
//   NC-Task 1 SAF/Axes/working2_open_bag <-> Place2/place2_openbag
//     Drive/Inputs/In/nDataIn1 <-> Inputs/Following error actual value
//     Drive/Inputs/In/nDataIn3[0] <-> Inputs/Torque actual value
//     Drive/Inputs/In/nDcOutputTime <-> InfoData/DcOutputShift
//     Drive/Inputs/In/nState1 <-> Inputs/Statusword
//     Drive/Inputs/In/nState2 <-> Inputs/Statusword @bit 8
//     Drive/Inputs/In/nState4 @bit 1 <-> WcState/InputToggle
//     Drive/Inputs/In/nState4 <-> WcState/WcState
//     Drive/Outputs/Out/nCtrl1 <-> Outputs/Controlword
//     Drive/Outputs/Out/nCtrl2 <-> Outputs/Controlword @bit 8
//     Drive/Outputs/Out/nDataOut1 <-> Outputs/Target position
//     Enc/Inputs/In/nDataIn1 <-> Inputs/Position actual value
//     Enc/Inputs/In/nDataIn3 <-> Inputs/Touch probe pos1 pos value
//     Enc/Inputs/In/nDataIn5 <-> Inputs/Touch probe pos2 pos value
//     Enc/Inputs/In/nDcInputTime <-> InfoData/DcInputShift
//     Enc/Inputs/In/nState4 @bit 1 <-> WcState/InputToggle
//     Enc/Inputs/In/nState4 <-> WcState/WcState
//     Enc/Inputs/In/nState5 <-> Inputs/Touch probe status
//     Enc/Inputs/In/nState6 <-> Inputs/Touch probe status @bit 8
//     Enc/Outputs/Out/nCtrl5 <-> Outputs/Touch probe function
//     Enc/Outputs/Out/nCtrl6 <-> Outputs/Touch probe function @bit 8
//   Rohlik_Expansion/Rohlik_Expansion Instance <-> Device 1 (EtherCAT Automation Protocol)
//     MianTask Inputs/G_IO.devState_Device1 <-> Inputs/DevState
//   Rohlik_Expansion/Rohlik_Expansion Instance <-> Lift
//     MianTask Inputs/G_IO.wcState_lift <-> Inputs/Frm0WcState
//   Rohlik_Expansion/Rohlik_Expansion Instance <-> Lift/Box 26 (ifm IO-Link Master AL1332)
//     MianTask Inputs/G_IO.arIOLinkQualifier_Lift/CH[{0..7}] <-> TxPDO IO-Link Port Qualifier/Qualifier of IO-Link Ch.{1..8}  (8 links)
//     MianTask Inputs/G_IO.arIOLinkTx_Lift[0]/InputByte[0] <-> Module 1 (IOL_4/4_I/O-Bytes)/TxPDO/input byte 0
//     MianTask Inputs/G_IO.arIOLinkTx_Lift[0]/InputByte[1] <-> Module 1 (IOL_4/4_I/O-Bytes)/TxPDO/input byte 1
//     MianTask Inputs/G_IO.arIOLinkTx_Lift[0]/InputByte[2] <-> Module 1 (IOL_4/4_I/O-Bytes)/TxPDO/input byte 2
//     MianTask Inputs/G_IO.arIOLinkTx_Lift[0]/InputByte[3] <-> Module 1 (IOL_4/4_I/O-Bytes)/TxPDO/input byte 3
//     MianTask Inputs/G_IO.arIOLinkTx_Lift[1]/InputByte[0] <-> Module 2 (IOL_4/4_I/O-Bytes)/TxPDO/input byte 0
//     MianTask Inputs/G_IO.arIOLinkTx_Lift[1]/InputByte[1] <-> Module 2 (IOL_4/4_I/O-Bytes)/TxPDO/input byte 1
//     MianTask Inputs/G_IO.arIOLinkTx_Lift[1]/InputByte[2] <-> Module 2 (IOL_4/4_I/O-Bytes)/TxPDO/input byte 2
//     MianTask Inputs/G_IO.arIOLinkTx_Lift[1]/InputByte[3] <-> Module 2 (IOL_4/4_I/O-Bytes)/TxPDO/input byte 3
//     MianTask Inputs/G_IO.arIOLinkTx_Lift[2]/InputByte[0] <-> Module 3 (IOL_4/4_I/O-Bytes)/TxPDO/input byte 0
//     MianTask Inputs/G_IO.arIOLinkTx_Lift[2]/InputByte[1] <-> Module 3 (IOL_4/4_I/O-Bytes)/TxPDO/input byte 1
//     MianTask Inputs/G_IO.arIOLinkTx_Lift[2]/InputByte[2] <-> Module 3 (IOL_4/4_I/O-Bytes)/TxPDO/input byte 2
//     MianTask Inputs/G_IO.arIOLinkTx_Lift[2]/InputByte[3] <-> Module 3 (IOL_4/4_I/O-Bytes)/TxPDO/input byte 3
//     MianTask Inputs/G_IO.arIOLinkTx_Lift[3]/InputByte[0] <-> Module 4 (IOL_4/4_I/O-Bytes)/TxPDO/input byte 0
//     MianTask Inputs/G_IO.arIOLinkTx_Lift[3]/InputByte[1] <-> Module 4 (IOL_4/4_I/O-Bytes)/TxPDO/input byte 1
//     MianTask Inputs/G_IO.arIOLinkTx_Lift[3]/InputByte[2] <-> Module 4 (IOL_4/4_I/O-Bytes)/TxPDO/input byte 2
//     MianTask Inputs/G_IO.arIOLinkTx_Lift[3]/InputByte[3] <-> Module 4 (IOL_4/4_I/O-Bytes)/TxPDO/input byte 3
//     MianTask Inputs/G_IO.arIOLinkTx_Lift[4]/InputByte[0] <-> Module 5 (IOL_4/4_I/O-Bytes)/TxPDO/input byte 0
//     MianTask Inputs/G_IO.arIOLinkTx_Lift[4]/InputByte[1] <-> Module 5 (IOL_4/4_I/O-Bytes)/TxPDO/input byte 1
//     MianTask Inputs/G_IO.arIOLinkTx_Lift[4]/InputByte[2] <-> Module 5 (IOL_4/4_I/O-Bytes)/TxPDO/input byte 2
//     MianTask Inputs/G_IO.arIOLinkTx_Lift[4]/InputByte[3] <-> Module 5 (IOL_4/4_I/O-Bytes)/TxPDO/input byte 3
//     MianTask Inputs/G_IO.arIOLinkTx_Lift[5]/InputByte[0] <-> Module 6 (IOL_4/4_I/O-Bytes)/TxPDO/input byte 0
//     MianTask Inputs/G_IO.arIOLinkTx_Lift[5]/InputByte[1] <-> Module 6 (IOL_4/4_I/O-Bytes)/TxPDO/input byte 1
//     MianTask Inputs/G_IO.arIOLinkTx_Lift[5]/InputByte[2] <-> Module 6 (IOL_4/4_I/O-Bytes)/TxPDO/input byte 2
//     MianTask Inputs/G_IO.arIOLinkTx_Lift[5]/InputByte[3] <-> Module 6 (IOL_4/4_I/O-Bytes)/TxPDO/input byte 3
//     MianTask Inputs/G_IO.arIOLinkTx_Lift[6]/InputByte[0] <-> Module 7 (IOL_4/4_I/O-Bytes)/TxPDO/input byte 0
//     MianTask Inputs/G_IO.arIOLinkTx_Lift[6]/InputByte[1] <-> Module 7 (IOL_4/4_I/O-Bytes)/TxPDO/input byte 1
//     MianTask Inputs/G_IO.arIOLinkTx_Lift[6]/InputByte[2] <-> Module 7 (IOL_4/4_I/O-Bytes)/TxPDO/input byte 2
//     MianTask Inputs/G_IO.arIOLinkTx_Lift[6]/InputByte[3] <-> Module 7 (IOL_4/4_I/O-Bytes)/TxPDO/input byte 3
//     MianTask Inputs/G_IO.arIOLinkTx_Lift[7]/InputByte[0] <-> Module 8 (IOL_4/4_I/O-Bytes)/TxPDO/input byte 0
//     MianTask Inputs/G_IO.arIOLinkTx_Lift[7]/InputByte[1] <-> Module 8 (IOL_4/4_I/O-Bytes)/TxPDO/input byte 1
//     MianTask Inputs/G_IO.arIOLinkTx_Lift[7]/InputByte[2] <-> Module 8 (IOL_4/4_I/O-Bytes)/TxPDO/input byte 2
//     MianTask Inputs/G_IO.arIOLinkTx_Lift[7]/InputByte[3] <-> Module 8 (IOL_4/4_I/O-Bytes)/TxPDO/input byte 3
//     MianTask Outputs/G_IO.arIOLinkRx_Lift[0]/OutputByte[0] <-> Module 1 (IOL_4/4_I/O-Bytes)/RxPDO/output byte 0
//     MianTask Outputs/G_IO.arIOLinkRx_Lift[0]/OutputByte[1] <-> Module 1 (IOL_4/4_I/O-Bytes)/RxPDO/output byte 1
//     MianTask Outputs/G_IO.arIOLinkRx_Lift[0]/OutputByte[2] <-> Module 1 (IOL_4/4_I/O-Bytes)/RxPDO/output byte 2
//     MianTask Outputs/G_IO.arIOLinkRx_Lift[0]/OutputByte[3] <-> Module 1 (IOL_4/4_I/O-Bytes)/RxPDO/output byte 3
//     MianTask Outputs/G_IO.arIOLinkRx_Lift[1]/OutputByte[0] <-> Module 2 (IOL_4/4_I/O-Bytes)/RxPDO/output byte 0
//     MianTask Outputs/G_IO.arIOLinkRx_Lift[1]/OutputByte[1] <-> Module 2 (IOL_4/4_I/O-Bytes)/RxPDO/output byte 1
//     MianTask Outputs/G_IO.arIOLinkRx_Lift[1]/OutputByte[2] <-> Module 2 (IOL_4/4_I/O-Bytes)/RxPDO/output byte 2
//     MianTask Outputs/G_IO.arIOLinkRx_Lift[1]/OutputByte[3] <-> Module 2 (IOL_4/4_I/O-Bytes)/RxPDO/output byte 3
//     MianTask Outputs/G_IO.arIOLinkRx_Lift[2]/OutputByte[0] <-> Module 3 (IOL_4/4_I/O-Bytes)/RxPDO/output byte 0
//     MianTask Outputs/G_IO.arIOLinkRx_Lift[2]/OutputByte[1] <-> Module 3 (IOL_4/4_I/O-Bytes)/RxPDO/output byte 1
//     MianTask Outputs/G_IO.arIOLinkRx_Lift[2]/OutputByte[2] <-> Module 3 (IOL_4/4_I/O-Bytes)/RxPDO/output byte 2
//     MianTask Outputs/G_IO.arIOLinkRx_Lift[2]/OutputByte[3] <-> Module 3 (IOL_4/4_I/O-Bytes)/RxPDO/output byte 3
//     MianTask Outputs/G_IO.arIOLinkRx_Lift[3]/OutputByte[0] <-> Module 4 (IOL_4/4_I/O-Bytes)/RxPDO/output byte 0
//     MianTask Outputs/G_IO.arIOLinkRx_Lift[3]/OutputByte[1] <-> Module 4 (IOL_4/4_I/O-Bytes)/RxPDO/output byte 1
//     MianTask Outputs/G_IO.arIOLinkRx_Lift[3]/OutputByte[2] <-> Module 4 (IOL_4/4_I/O-Bytes)/RxPDO/output byte 2
//     MianTask Outputs/G_IO.arIOLinkRx_Lift[3]/OutputByte[3] <-> Module 4 (IOL_4/4_I/O-Bytes)/RxPDO/output byte 3
//     MianTask Outputs/G_IO.arIOLinkRx_Lift[4]/OutputByte[0] <-> Module 5 (IOL_4/4_I/O-Bytes)/RxPDO/output byte 0
//     MianTask Outputs/G_IO.arIOLinkRx_Lift[4]/OutputByte[1] <-> Module 5 (IOL_4/4_I/O-Bytes)/RxPDO/output byte 1
//     MianTask Outputs/G_IO.arIOLinkRx_Lift[4]/OutputByte[2] <-> Module 5 (IOL_4/4_I/O-Bytes)/RxPDO/output byte 2
//     MianTask Outputs/G_IO.arIOLinkRx_Lift[4]/OutputByte[3] <-> Module 5 (IOL_4/4_I/O-Bytes)/RxPDO/output byte 3
//     MianTask Outputs/G_IO.arIOLinkRx_Lift[5]/OutputByte[0] <-> Module 6 (IOL_4/4_I/O-Bytes)/RxPDO/output byte 0
//     MianTask Outputs/G_IO.arIOLinkRx_Lift[5]/OutputByte[1] <-> Module 6 (IOL_4/4_I/O-Bytes)/RxPDO/output byte 1
//     MianTask Outputs/G_IO.arIOLinkRx_Lift[5]/OutputByte[2] <-> Module 6 (IOL_4/4_I/O-Bytes)/RxPDO/output byte 2
//     MianTask Outputs/G_IO.arIOLinkRx_Lift[5]/OutputByte[3] <-> Module 6 (IOL_4/4_I/O-Bytes)/RxPDO/output byte 3
//     MianTask Outputs/G_IO.arIOLinkRx_Lift[6]/OutputByte[0] <-> Module 7 (IOL_4/4_I/O-Bytes)/RxPDO/output byte 0
//     MianTask Outputs/G_IO.arIOLinkRx_Lift[6]/OutputByte[1] <-> Module 7 (IOL_4/4_I/O-Bytes)/RxPDO/output byte 1
//     MianTask Outputs/G_IO.arIOLinkRx_Lift[6]/OutputByte[2] <-> Module 7 (IOL_4/4_I/O-Bytes)/RxPDO/output byte 2
//     MianTask Outputs/G_IO.arIOLinkRx_Lift[6]/OutputByte[3] <-> Module 7 (IOL_4/4_I/O-Bytes)/RxPDO/output byte 3
//     MianTask Outputs/G_IO.arIOLinkRx_Lift[7]/OutputByte[0] <-> Module 8 (IOL_4/4_I/O-Bytes)/RxPDO/output byte 0
//     MianTask Outputs/G_IO.arIOLinkRx_Lift[7]/OutputByte[1] <-> Module 8 (IOL_4/4_I/O-Bytes)/RxPDO/output byte 1
//     MianTask Outputs/G_IO.arIOLinkRx_Lift[7]/OutputByte[2] <-> Module 8 (IOL_4/4_I/O-Bytes)/RxPDO/output byte 2
//     MianTask Outputs/G_IO.arIOLinkRx_Lift[7]/OutputByte[3] <-> Module 8 (IOL_4/4_I/O-Bytes)/RxPDO/output byte 3
//   Rohlik_Expansion/Rohlik_Expansion Instance <-> Lift/Term 17 (EK1100)/DI2
//     MianTask Inputs/G_IO.arDI[2]/Ch[{0..15}] <-> Channel {1..16}/Input  (16 links)
//   Rohlik_Expansion/Rohlik_Expansion Instance <-> Lift/Term 17 (EK1100)/DI3
//     MianTask Inputs/G_IO.arDI[3]/Ch[{0..15}] <-> Channel {1..16}/Input  (16 links)
//   Rohlik_Expansion/Rohlik_Expansion Instance <-> Lift/Term 17 (EK1100)/DO2
//     MianTask Outputs/G_IO.arDO[2]/Ch[{0..15}] <-> Channel {1..16}/Output  (16 links)
//   Rohlik_Expansion/Rohlik_Expansion Instance <-> Lift/Term 17 (EK1100)/DO3
//     MianTask Outputs/G_IO.arDO[3]/Ch[{0..15}] <-> Channel {1..16}/Output  (16 links)
//   Rohlik_Expansion/Rohlik_Expansion Instance <-> Lift/Term 17 (EK1100)/SI4
//     MianTask Inputs/G_IO.arSI[4]/Ch[{1..4}] <-> Module 1 (FSOES)/TxPDO/FSOE/InputChannel{1..4}  (4 links)
//   Rohlik_Expansion/Rohlik_Expansion Instance <-> Lift/Term 17 (EK1100)/SI5
//     MianTask Inputs/G_IO.arSI[5]/Ch[{1..4}] <-> Module 1 (FSOES)/TxPDO/FSOE/InputChannel{1..4}  (4 links)
//   Rohlik_Expansion/Rohlik_Expansion Instance <-> Lift/Term 17 (EK1100)/SI6
//     MianTask Inputs/G_IO.arSI[6]/Ch[{1..4}] <-> Module 1 (FSOES)/TxPDO/FSOE/InputChannel{1..4}  (4 links)
//   Rohlik_Expansion/Rohlik_Expansion Instance <-> MCP
//     MianTask Inputs/G_IO.wcState_mcp <-> Inputs/Frm0WcState
//   Rohlik_Expansion/Rohlik_Expansion Instance <-> MCP/MCP-EK1100/DI0
//     MianTask Inputs/G_IO.arDI[0]/Ch[{0..15}] <-> Channel {1..16}/Input  (16 links)
//   Rohlik_Expansion/Rohlik_Expansion Instance <-> MCP/MCP-EK1100/DI1
//     MianTask Inputs/G_IO.arDI[1]/Ch[{0..15}] <-> Channel {1..16}/Input  (16 links)
//   Rohlik_Expansion/Rohlik_Expansion Instance <-> MCP/MCP-EK1100/DO0
//     MianTask Outputs/G_IO.arDO[0]/Ch[{0..15}] <-> Channel {1..16}/Output  (16 links)
//   Rohlik_Expansion/Rohlik_Expansion Instance <-> MCP/MCP-EK1100/DO1
//     MianTask Outputs/G_IO.arDO[1]/Ch[{0..15}] <-> Channel {1..16}/Output  (16 links)
//   Rohlik_Expansion/Rohlik_Expansion Instance <-> MCP/MCP-EK1100/SI0
//     MianTask Inputs/G_IO.arSI[0]/Ch[{1..4}] <-> Module 1 (FSOES)/TxPDO/FSOE/InputChannel{1..4}  (4 links)
//   Rohlik_Expansion/Rohlik_Expansion Instance <-> MCP/MCP-EK1100/SI1
//     MianTask Inputs/G_IO.arSI[1]/Ch[{1..4}] <-> Module 1 (FSOES)/TxPDO/FSOE/InputChannel{1..4}  (4 links)
//   Rohlik_Expansion/Rohlik_Expansion Instance <-> MCP/MCP-EK1100/SI2
//     MianTask Inputs/G_IO.arSI[2]/Ch[{1..4}] <-> Module 1 (FSOES)/TxPDO/FSOE/InputChannel{1..4}  (4 links)
//   Rohlik_Expansion/Rohlik_Expansion Instance <-> MCP/MCP-EK1100/SI3
//     MianTask Inputs/G_IO.arSI[3]/Ch[{1..4}] <-> Module 1 (FSOES)/TxPDO/FSOE/InputChannel{1..4}  (4 links)
//   Rohlik_Expansion/Rohlik_Expansion Instance <-> MCP/MCP-EK1100/SI7
//     MianTask Inputs/G_IO.arSI[7]/Ch[{1..4}] <-> Module 1 (FSOES)/TxPDO/FSOE/InputChannel{1..4}  (4 links)
//   Rohlik_Expansion/Rohlik_Expansion Instance <-> MCP/MCP-EK1100/SI8
//     MianTask Inputs/G_IO.arSI[8]/Ch[{1..4}] <-> Module 1 (FSOES)/TxPDO/FSOE/InputChannel{1..4}  (4 links)
//   Rohlik_Expansion/Rohlik_Expansion Instance <-> MCP/MCP-EK1100/Term 13 (EL3064)
//     MianTask Inputs/GVL.iAng_AirFlow_left <-> AI Standard Channel 3/Value
//     MianTask Inputs/GVL.iAng_AirFlow_right <-> AI Standard Channel 4/Value
//     MianTask Inputs/GVL.iAng_airPress_left <-> AI Standard Channel 1/Value
//     MianTask Inputs/GVL.iAng_airPress_right <-> AI Standard Channel 2/Value
//   Rohlik_Expansion/Rohlik_Expansion Instance <-> MCP/MCP-EK1100/Term 7 (EL6910)
//     MianTask Inputs/GVL_SAFETY.Lift_STO <-> StandardInputs/Standard Out Var 42
//     MianTask Inputs/GVL_SAFETY.Place1_STO <-> StandardInputs/Standard Out Var 43
//     MianTask Inputs/GVL_SAFETY.Place2_STO <-> StandardInputs/Standard Out Var 44
//     MianTask Inputs/GVL_SAFETY.SO0_0 <-> StandardInputs/Standard Out Var 45
//     MianTask Inputs/GVL_SAFETY.SO0_1 <-> StandardInputs/Standard Out Var 47
//     MianTask Inputs/GVL_SAFETY.SO0_2 <-> StandardInputs/Standard Out Var 46
//     MianTask Inputs/GVL_SAFETY.SO0_3 <-> StandardInputs/Standard Out Var 48
//     MianTask Inputs/GVL_SAFETY.SO1_0 <-> StandardInputs/Standard Out Var 42
//     MianTask Inputs/GVL_SAFETY.SO1_1 <-> StandardInputs/Standard Out Var 43
//     MianTask Inputs/GVL_SAFETY.SO1_2 <-> StandardInputs/Standard Out Var 44
//     MianTask Inputs/GVL_SAFETY.SO2_0 <-> StandardInputs/Standard Out Var 42
//     MianTask Inputs/GVL_SAFETY.SO2_1 <-> StandardInputs/Standard Out Var 43
//     MianTask Inputs/GVL_SAFETY.SO2_2 <-> StandardInputs/Standard Out Var 44
//     MianTask Inputs/GVL_SAFETY.SO3_0 <-> StandardInputs/Standard Out Var 42
//     MianTask Inputs/GVL_SAFETY.SO3_1 <-> StandardInputs/Standard Out Var 43
//     MianTask Inputs/GVL_SAFETY.SO3_2 <-> StandardInputs/Standard Out Var 44
//     MianTask Inputs/GVL_SAFETY.SO4_0 <-> StandardInputs/Standard Out Var 59
//     MianTask Inputs/GVL_SAFETY.SO4_1 <-> StandardInputs/Standard Out Var 60
//     MianTask Inputs/GVL_SAFETY.bAirDump1 <-> StandardInputs/Standard Out Var 77
//     MianTask Inputs/GVL_SAFETY.bAirDump2 <-> StandardInputs/Standard Out Var 78
//     MianTask Inputs/GVL_SAFETY.b_ComError <-> StandardInputs/Standard Out Var 18
//     MianTask Inputs/GVL_SAFETY.b_FBerror <-> StandardInputs/Standard Out Var 19
//     MianTask Inputs/GVL_SAFETY.robot1_STO_EAS <-> StandardInputs/Standard Out Var 47
//     MianTask Inputs/GVL_SAFETY.robot2_STO_EAS <-> StandardInputs/Standard Out Var 48
//     MianTask Inputs/GVL_SAFETY.robot1_STO_EES <-> StandardInputs/Standard Out Var 45
//     MianTask Inputs/GVL_SAFETY.robot2_STO_EES <-> StandardInputs/Standard Out Var 46
//     MianTask Outputs/GVL_SAFETY.bLeftDoorUnlock_Request <-> StandardOutputs/Standard In Var 34
//     MianTask Outputs/GVL_SAFETY.bRightDoorUnlock_Request <-> StandardOutputs/Standard In Var 35
//     MianTask Outputs/GVL_SAFETY.bSafetyReset_airDump <-> StandardOutputs/Standard In Var 73
//     MianTask Outputs/GVL_SAFETY.bSafetyRestart_left <-> StandardOutputs/Standard In Var 65
//     MianTask Outputs/GVL_SAFETY.bSafetyRestart_right <-> StandardOutputs/Standard In Var 66
//     MianTask Outputs/GVL_SAFETY.b_EStopRestart <-> StandardOutputs/Standard In Var 16
//     MianTask Outputs/GVL_SAFETY.b_ErrorAck <-> StandardOutputs/Standard In Var 15
//     MianTask Outputs/GVL_SAFETY.b_GroupRun <-> StandardOutputs/Standard In Var 14
//   Rohlik_Expansion/Rohlik_Expansion Instance <-> Place1
//     MianTask Inputs/G_IO.wcState_place1 <-> Inputs/Frm0WcState
//   Rohlik_Expansion/Rohlik_Expansion Instance <-> Place1/Box 36 (ifm IO-Link Master AL1332)
//     MianTask Inputs/G_IO.arIOLinkQualifier_Place1/CH[{0..7}] <-> TxPDO IO-Link Port Qualifier/Qualifier of IO-Link Ch.{1..8}  (8 links)
//     MianTask Inputs/G_IO.arIOLinkTx_Place1[0]/InputByte[0] <-> Module 1 (IOL_4/4_I/O-Bytes)/TxPDO/input byte 0
//     MianTask Inputs/G_IO.arIOLinkTx_Place1[0]/InputByte[1] <-> Module 1 (IOL_4/4_I/O-Bytes)/TxPDO/input byte 1
//     MianTask Inputs/G_IO.arIOLinkTx_Place1[0]/InputByte[2] <-> Module 1 (IOL_4/4_I/O-Bytes)/TxPDO/input byte 2
//     MianTask Inputs/G_IO.arIOLinkTx_Place1[0]/InputByte[3] <-> Module 1 (IOL_4/4_I/O-Bytes)/TxPDO/input byte 3
//     MianTask Inputs/G_IO.arIOLinkTx_Place1[1]/InputByte[0] <-> Module 2 (IOL_4/4_I/O-Bytes)/TxPDO/input byte 0
//     MianTask Inputs/G_IO.arIOLinkTx_Place1[1]/InputByte[1] <-> Module 2 (IOL_4/4_I/O-Bytes)/TxPDO/input byte 1
//     MianTask Inputs/G_IO.arIOLinkTx_Place1[1]/InputByte[2] <-> Module 2 (IOL_4/4_I/O-Bytes)/TxPDO/input byte 2
//     MianTask Inputs/G_IO.arIOLinkTx_Place1[1]/InputByte[3] <-> Module 2 (IOL_4/4_I/O-Bytes)/TxPDO/input byte 3
//     MianTask Inputs/G_IO.arIOLinkTx_Place1[2]/InputByte[0] <-> Module 3 (IOL_4/4_I/O-Bytes)/TxPDO/input byte 0
//     MianTask Inputs/G_IO.arIOLinkTx_Place1[2]/InputByte[1] <-> Module 3 (IOL_4/4_I/O-Bytes)/TxPDO/input byte 1
//     MianTask Inputs/G_IO.arIOLinkTx_Place1[2]/InputByte[2] <-> Module 3 (IOL_4/4_I/O-Bytes)/TxPDO/input byte 2
//     MianTask Inputs/G_IO.arIOLinkTx_Place1[2]/InputByte[3] <-> Module 3 (IOL_4/4_I/O-Bytes)/TxPDO/input byte 3
//     MianTask Inputs/G_IO.arIOLinkTx_Place1[3]/InputByte[0] <-> Module 4 (IOL_4/4_I/O-Bytes)/TxPDO/input byte 0
//     MianTask Inputs/G_IO.arIOLinkTx_Place1[3]/InputByte[1] <-> Module 4 (IOL_4/4_I/O-Bytes)/TxPDO/input byte 1
//     MianTask Inputs/G_IO.arIOLinkTx_Place1[3]/InputByte[2] <-> Module 4 (IOL_4/4_I/O-Bytes)/TxPDO/input byte 2
//     MianTask Inputs/G_IO.arIOLinkTx_Place1[3]/InputByte[3] <-> Module 4 (IOL_4/4_I/O-Bytes)/TxPDO/input byte 3
//     MianTask Inputs/G_IO.arIOLinkTx_Place1[4]/InputByte[0] <-> Module 5 (IOL_4/4_I/O-Bytes)/TxPDO/input byte 0
//     MianTask Inputs/G_IO.arIOLinkTx_Place1[4]/InputByte[1] <-> Module 5 (IOL_4/4_I/O-Bytes)/TxPDO/input byte 1
//     MianTask Inputs/G_IO.arIOLinkTx_Place1[4]/InputByte[2] <-> Module 5 (IOL_4/4_I/O-Bytes)/TxPDO/input byte 2
//     MianTask Inputs/G_IO.arIOLinkTx_Place1[4]/InputByte[3] <-> Module 5 (IOL_4/4_I/O-Bytes)/TxPDO/input byte 3
//     MianTask Inputs/G_IO.arIOLinkTx_Place1[5]/InputByte[0] <-> Module 6 (IOL_4/4_I/O-Bytes)/TxPDO/input byte 0
//     MianTask Inputs/G_IO.arIOLinkTx_Place1[5]/InputByte[1] <-> Module 6 (IOL_4/4_I/O-Bytes)/TxPDO/input byte 1
//     MianTask Inputs/G_IO.arIOLinkTx_Place1[5]/InputByte[2] <-> Module 6 (IOL_4/4_I/O-Bytes)/TxPDO/input byte 2
//     MianTask Inputs/G_IO.arIOLinkTx_Place1[5]/InputByte[3] <-> Module 6 (IOL_4/4_I/O-Bytes)/TxPDO/input byte 3
//     MianTask Inputs/G_IO.arIOLinkTx_Place1[6]/InputByte[0] <-> Module 7 (IOL_4/4_I/O-Bytes)/TxPDO/input byte 0
//     MianTask Inputs/G_IO.arIOLinkTx_Place1[6]/InputByte[1] <-> Module 7 (IOL_4/4_I/O-Bytes)/TxPDO/input byte 1
//     MianTask Inputs/G_IO.arIOLinkTx_Place1[6]/InputByte[2] <-> Module 7 (IOL_4/4_I/O-Bytes)/TxPDO/input byte 2
//     MianTask Inputs/G_IO.arIOLinkTx_Place1[6]/InputByte[3] <-> Module 7 (IOL_4/4_I/O-Bytes)/TxPDO/input byte 3
//     MianTask Inputs/G_IO.arIOLinkTx_Place1[7]/InputByte[0] <-> Module 8 (IOL_4/4_I/O-Bytes)/TxPDO/input byte 0
//     MianTask Inputs/G_IO.arIOLinkTx_Place1[7]/InputByte[1] <-> Module 8 (IOL_4/4_I/O-Bytes)/TxPDO/input byte 1
//     MianTask Inputs/G_IO.arIOLinkTx_Place1[7]/InputByte[2] <-> Module 8 (IOL_4/4_I/O-Bytes)/TxPDO/input byte 2
//     MianTask Inputs/G_IO.arIOLinkTx_Place1[7]/InputByte[3] <-> Module 8 (IOL_4/4_I/O-Bytes)/TxPDO/input byte 3
//     MianTask Outputs/G_IO.arIOLinkRx_Place1[0]/OutputByte[0] <-> Module 1 (IOL_4/4_I/O-Bytes)/RxPDO/output byte 0
//     MianTask Outputs/G_IO.arIOLinkRx_Place1[0]/OutputByte[1] <-> Module 1 (IOL_4/4_I/O-Bytes)/RxPDO/output byte 1
//     MianTask Outputs/G_IO.arIOLinkRx_Place1[0]/OutputByte[2] <-> Module 1 (IOL_4/4_I/O-Bytes)/RxPDO/output byte 2
//     MianTask Outputs/G_IO.arIOLinkRx_Place1[0]/OutputByte[3] <-> Module 1 (IOL_4/4_I/O-Bytes)/RxPDO/output byte 3
//     MianTask Outputs/G_IO.arIOLinkRx_Place1[1]/OutputByte[0] <-> Module 2 (IOL_4/4_I/O-Bytes)/RxPDO/output byte 0
//     MianTask Outputs/G_IO.arIOLinkRx_Place1[1]/OutputByte[1] <-> Module 2 (IOL_4/4_I/O-Bytes)/RxPDO/output byte 1
//     MianTask Outputs/G_IO.arIOLinkRx_Place1[1]/OutputByte[2] <-> Module 2 (IOL_4/4_I/O-Bytes)/RxPDO/output byte 2
//     MianTask Outputs/G_IO.arIOLinkRx_Place1[1]/OutputByte[3] <-> Module 2 (IOL_4/4_I/O-Bytes)/RxPDO/output byte 3
//     MianTask Outputs/G_IO.arIOLinkRx_Place1[2]/OutputByte[0] <-> Module 3 (IOL_4/4_I/O-Bytes)/RxPDO/output byte 0
//     MianTask Outputs/G_IO.arIOLinkRx_Place1[2]/OutputByte[1] <-> Module 3 (IOL_4/4_I/O-Bytes)/RxPDO/output byte 1
//     MianTask Outputs/G_IO.arIOLinkRx_Place1[2]/OutputByte[2] <-> Module 3 (IOL_4/4_I/O-Bytes)/RxPDO/output byte 2
//     MianTask Outputs/G_IO.arIOLinkRx_Place1[2]/OutputByte[3] <-> Module 3 (IOL_4/4_I/O-Bytes)/RxPDO/output byte 3
//     MianTask Outputs/G_IO.arIOLinkRx_Place1[3]/OutputByte[0] <-> Module 4 (IOL_4/4_I/O-Bytes)/RxPDO/output byte 0
//     MianTask Outputs/G_IO.arIOLinkRx_Place1[3]/OutputByte[1] <-> Module 4 (IOL_4/4_I/O-Bytes)/RxPDO/output byte 1
//     MianTask Outputs/G_IO.arIOLinkRx_Place1[3]/OutputByte[2] <-> Module 4 (IOL_4/4_I/O-Bytes)/RxPDO/output byte 2
//     MianTask Outputs/G_IO.arIOLinkRx_Place1[3]/OutputByte[3] <-> Module 4 (IOL_4/4_I/O-Bytes)/RxPDO/output byte 3
//     MianTask Outputs/G_IO.arIOLinkRx_Place1[4]/OutputByte[0] <-> Module 5 (IOL_4/4_I/O-Bytes)/RxPDO/output byte 0
//     MianTask Outputs/G_IO.arIOLinkRx_Place1[4]/OutputByte[1] <-> Module 5 (IOL_4/4_I/O-Bytes)/RxPDO/output byte 1
//     MianTask Outputs/G_IO.arIOLinkRx_Place1[4]/OutputByte[2] <-> Module 5 (IOL_4/4_I/O-Bytes)/RxPDO/output byte 2
//     MianTask Outputs/G_IO.arIOLinkRx_Place1[4]/OutputByte[3] <-> Module 5 (IOL_4/4_I/O-Bytes)/RxPDO/output byte 3
//     MianTask Outputs/G_IO.arIOLinkRx_Place1[5]/OutputByte[0] <-> Module 6 (IOL_4/4_I/O-Bytes)/RxPDO/output byte 0
//     MianTask Outputs/G_IO.arIOLinkRx_Place1[5]/OutputByte[1] <-> Module 6 (IOL_4/4_I/O-Bytes)/RxPDO/output byte 1
//     MianTask Outputs/G_IO.arIOLinkRx_Place1[5]/OutputByte[2] <-> Module 6 (IOL_4/4_I/O-Bytes)/RxPDO/output byte 2
//     MianTask Outputs/G_IO.arIOLinkRx_Place1[5]/OutputByte[3] <-> Module 6 (IOL_4/4_I/O-Bytes)/RxPDO/output byte 3
//     MianTask Outputs/G_IO.arIOLinkRx_Place1[6]/OutputByte[0] <-> Module 7 (IOL_4/4_I/O-Bytes)/RxPDO/output byte 0
//     MianTask Outputs/G_IO.arIOLinkRx_Place1[6]/OutputByte[1] <-> Module 7 (IOL_4/4_I/O-Bytes)/RxPDO/output byte 1
//     MianTask Outputs/G_IO.arIOLinkRx_Place1[6]/OutputByte[2] <-> Module 7 (IOL_4/4_I/O-Bytes)/RxPDO/output byte 2
//     MianTask Outputs/G_IO.arIOLinkRx_Place1[6]/OutputByte[3] <-> Module 7 (IOL_4/4_I/O-Bytes)/RxPDO/output byte 3
//     MianTask Outputs/G_IO.arIOLinkRx_Place1[7]/OutputByte[0] <-> Module 8 (IOL_4/4_I/O-Bytes)/RxPDO/output byte 0
//     MianTask Outputs/G_IO.arIOLinkRx_Place1[7]/OutputByte[1] <-> Module 8 (IOL_4/4_I/O-Bytes)/RxPDO/output byte 1
//     MianTask Outputs/G_IO.arIOLinkRx_Place1[7]/OutputByte[2] <-> Module 8 (IOL_4/4_I/O-Bytes)/RxPDO/output byte 2
//     MianTask Outputs/G_IO.arIOLinkRx_Place1[7]/OutputByte[3] <-> Module 8 (IOL_4/4_I/O-Bytes)/RxPDO/output byte 3
//   Rohlik_Expansion/Rohlik_Expansion Instance <-> Place1/Term 27 (EK1100)/DI4
//     MianTask Inputs/G_IO.arDI[4]/Ch[{0..15}] <-> Channel {1..16}/Input  (16 links)
//   Rohlik_Expansion/Rohlik_Expansion Instance <-> Place1/Term 27 (EK1100)/DI5
//     MianTask Inputs/G_IO.arDI[5]/Ch[{0..15}] <-> Channel {1..16}/Input  (16 links)
//   Rohlik_Expansion/Rohlik_Expansion Instance <-> Place1/Term 27 (EK1100)/DO4
//     MianTask Outputs/G_IO.arDO[4]/Ch[{0..15}] <-> Channel {1..16}/Output  (16 links)
//   Rohlik_Expansion/Rohlik_Expansion Instance <-> Place1/Term 27 (EK1100)/DO6
//     MianTask Outputs/G_IO.arDO[6]/Ch[{0..15}] <-> Channel {1..16}/Output  (16 links)
//   Rohlik_Expansion/Rohlik_Expansion Instance <-> Place2
//     MianTask Inputs/G_IO.wcState_place2 <-> Inputs/Frm0WcState
//   Rohlik_Expansion/Rohlik_Expansion Instance <-> Place2/Box 46 (ifm IO-Link Master AL1332)
//     MianTask Inputs/G_IO.arIOLinkQualifier_Place2/CH[{0..7}] <-> TxPDO IO-Link Port Qualifier/Qualifier of IO-Link Ch.{1..8}  (8 links)
//     MianTask Inputs/G_IO.arIOLinkTx_Place2[0]/InputByte[0] <-> Module 1 (IOL_4/4_I/O-Bytes)/TxPDO/input byte 0
//     MianTask Inputs/G_IO.arIOLinkTx_Place2[0]/InputByte[1] <-> Module 1 (IOL_4/4_I/O-Bytes)/TxPDO/input byte 1
//     MianTask Inputs/G_IO.arIOLinkTx_Place2[0]/InputByte[2] <-> Module 1 (IOL_4/4_I/O-Bytes)/TxPDO/input byte 2
//     MianTask Inputs/G_IO.arIOLinkTx_Place2[0]/InputByte[3] <-> Module 1 (IOL_4/4_I/O-Bytes)/TxPDO/input byte 3
//     MianTask Inputs/G_IO.arIOLinkTx_Place2[1]/InputByte[0] <-> Module 2 (IOL_4/4_I/O-Bytes)/TxPDO/input byte 0
//     MianTask Inputs/G_IO.arIOLinkTx_Place2[1]/InputByte[1] <-> Module 2 (IOL_4/4_I/O-Bytes)/TxPDO/input byte 1
//     MianTask Inputs/G_IO.arIOLinkTx_Place2[1]/InputByte[2] <-> Module 2 (IOL_4/4_I/O-Bytes)/TxPDO/input byte 2
//     MianTask Inputs/G_IO.arIOLinkTx_Place2[1]/InputByte[3] <-> Module 2 (IOL_4/4_I/O-Bytes)/TxPDO/input byte 3
//     MianTask Inputs/G_IO.arIOLinkTx_Place2[2]/InputByte[0] <-> Module 3 (IOL_4/4_I/O-Bytes)/TxPDO/input byte 0
//     MianTask Inputs/G_IO.arIOLinkTx_Place2[2]/InputByte[1] <-> Module 3 (IOL_4/4_I/O-Bytes)/TxPDO/input byte 1
//     MianTask Inputs/G_IO.arIOLinkTx_Place2[2]/InputByte[2] <-> Module 3 (IOL_4/4_I/O-Bytes)/TxPDO/input byte 2
//     MianTask Inputs/G_IO.arIOLinkTx_Place2[2]/InputByte[3] <-> Module 3 (IOL_4/4_I/O-Bytes)/TxPDO/input byte 3
//     MianTask Inputs/G_IO.arIOLinkTx_Place2[3]/InputByte[0] <-> Module 4 (IOL_4/4_I/O-Bytes)/TxPDO/input byte 0
//     MianTask Inputs/G_IO.arIOLinkTx_Place2[3]/InputByte[1] <-> Module 4 (IOL_4/4_I/O-Bytes)/TxPDO/input byte 1
//     MianTask Inputs/G_IO.arIOLinkTx_Place2[3]/InputByte[2] <-> Module 4 (IOL_4/4_I/O-Bytes)/TxPDO/input byte 2
//     MianTask Inputs/G_IO.arIOLinkTx_Place2[3]/InputByte[3] <-> Module 4 (IOL_4/4_I/O-Bytes)/TxPDO/input byte 3
//     MianTask Inputs/G_IO.arIOLinkTx_Place2[4]/InputByte[0] <-> Module 5 (IOL_4/4_I/O-Bytes)/TxPDO/input byte 0
//     MianTask Inputs/G_IO.arIOLinkTx_Place2[4]/InputByte[1] <-> Module 5 (IOL_4/4_I/O-Bytes)/TxPDO/input byte 1
//     MianTask Inputs/G_IO.arIOLinkTx_Place2[4]/InputByte[2] <-> Module 5 (IOL_4/4_I/O-Bytes)/TxPDO/input byte 2
//     MianTask Inputs/G_IO.arIOLinkTx_Place2[4]/InputByte[3] <-> Module 5 (IOL_4/4_I/O-Bytes)/TxPDO/input byte 3
//     MianTask Inputs/G_IO.arIOLinkTx_Place2[5]/InputByte[0] <-> Module 6 (IOL_4/4_I/O-Bytes)/TxPDO/input byte 0
//     MianTask Inputs/G_IO.arIOLinkTx_Place2[5]/InputByte[1] <-> Module 6 (IOL_4/4_I/O-Bytes)/TxPDO/input byte 1
//     MianTask Inputs/G_IO.arIOLinkTx_Place2[5]/InputByte[2] <-> Module 6 (IOL_4/4_I/O-Bytes)/TxPDO/input byte 2
//     MianTask Inputs/G_IO.arIOLinkTx_Place2[5]/InputByte[3] <-> Module 6 (IOL_4/4_I/O-Bytes)/TxPDO/input byte 3
//     MianTask Inputs/G_IO.arIOLinkTx_Place2[6]/InputByte[0] <-> Module 7 (IOL_4/4_I/O-Bytes)/TxPDO/input byte 0
//     MianTask Inputs/G_IO.arIOLinkTx_Place2[6]/InputByte[1] <-> Module 7 (IOL_4/4_I/O-Bytes)/TxPDO/input byte 1
//     MianTask Inputs/G_IO.arIOLinkTx_Place2[6]/InputByte[2] <-> Module 7 (IOL_4/4_I/O-Bytes)/TxPDO/input byte 2
//     MianTask Inputs/G_IO.arIOLinkTx_Place2[6]/InputByte[3] <-> Module 7 (IOL_4/4_I/O-Bytes)/TxPDO/input byte 3
//     MianTask Inputs/G_IO.arIOLinkTx_Place2[7]/InputByte[0] <-> Module 8 (IOL_4/4_I/O-Bytes)/TxPDO/input byte 0
//     MianTask Inputs/G_IO.arIOLinkTx_Place2[7]/InputByte[1] <-> Module 8 (IOL_4/4_I/O-Bytes)/TxPDO/input byte 1
//     MianTask Inputs/G_IO.arIOLinkTx_Place2[7]/InputByte[2] <-> Module 8 (IOL_4/4_I/O-Bytes)/TxPDO/input byte 2
//     MianTask Inputs/G_IO.arIOLinkTx_Place2[7]/InputByte[3] <-> Module 8 (IOL_4/4_I/O-Bytes)/TxPDO/input byte 3
//     MianTask Outputs/G_IO.arIOLinkRx_Place2[0]/OutputByte[0] <-> Module 1 (IOL_4/4_I/O-Bytes)/RxPDO/output byte 0
//     MianTask Outputs/G_IO.arIOLinkRx_Place2[0]/OutputByte[1] <-> Module 1 (IOL_4/4_I/O-Bytes)/RxPDO/output byte 1
//     MianTask Outputs/G_IO.arIOLinkRx_Place2[0]/OutputByte[2] <-> Module 1 (IOL_4/4_I/O-Bytes)/RxPDO/output byte 2
//     MianTask Outputs/G_IO.arIOLinkRx_Place2[0]/OutputByte[3] <-> Module 1 (IOL_4/4_I/O-Bytes)/RxPDO/output byte 3
//     MianTask Outputs/G_IO.arIOLinkRx_Place2[1]/OutputByte[0] <-> Module 2 (IOL_4/4_I/O-Bytes)/RxPDO/output byte 0
//     MianTask Outputs/G_IO.arIOLinkRx_Place2[1]/OutputByte[1] <-> Module 2 (IOL_4/4_I/O-Bytes)/RxPDO/output byte 1
//     MianTask Outputs/G_IO.arIOLinkRx_Place2[1]/OutputByte[2] <-> Module 2 (IOL_4/4_I/O-Bytes)/RxPDO/output byte 2
//     MianTask Outputs/G_IO.arIOLinkRx_Place2[1]/OutputByte[3] <-> Module 2 (IOL_4/4_I/O-Bytes)/RxPDO/output byte 3
//     MianTask Outputs/G_IO.arIOLinkRx_Place2[2]/OutputByte[0] <-> Module 3 (IOL_4/4_I/O-Bytes)/RxPDO/output byte 0
//     MianTask Outputs/G_IO.arIOLinkRx_Place2[2]/OutputByte[1] <-> Module 3 (IOL_4/4_I/O-Bytes)/RxPDO/output byte 1
//     MianTask Outputs/G_IO.arIOLinkRx_Place2[2]/OutputByte[2] <-> Module 3 (IOL_4/4_I/O-Bytes)/RxPDO/output byte 2
//     MianTask Outputs/G_IO.arIOLinkRx_Place2[2]/OutputByte[3] <-> Module 3 (IOL_4/4_I/O-Bytes)/RxPDO/output byte 3
//     MianTask Outputs/G_IO.arIOLinkRx_Place2[3]/OutputByte[0] <-> Module 4 (IOL_4/4_I/O-Bytes)/RxPDO/output byte 0
//     MianTask Outputs/G_IO.arIOLinkRx_Place2[3]/OutputByte[1] <-> Module 4 (IOL_4/4_I/O-Bytes)/RxPDO/output byte 1
//     MianTask Outputs/G_IO.arIOLinkRx_Place2[3]/OutputByte[2] <-> Module 4 (IOL_4/4_I/O-Bytes)/RxPDO/output byte 2
//     MianTask Outputs/G_IO.arIOLinkRx_Place2[3]/OutputByte[3] <-> Module 4 (IOL_4/4_I/O-Bytes)/RxPDO/output byte 3
//     MianTask Outputs/G_IO.arIOLinkRx_Place2[4]/OutputByte[0] <-> Module 5 (IOL_4/4_I/O-Bytes)/RxPDO/output byte 0
//     MianTask Outputs/G_IO.arIOLinkRx_Place2[4]/OutputByte[1] <-> Module 5 (IOL_4/4_I/O-Bytes)/RxPDO/output byte 1
//     MianTask Outputs/G_IO.arIOLinkRx_Place2[4]/OutputByte[2] <-> Module 5 (IOL_4/4_I/O-Bytes)/RxPDO/output byte 2
//     MianTask Outputs/G_IO.arIOLinkRx_Place2[4]/OutputByte[3] <-> Module 5 (IOL_4/4_I/O-Bytes)/RxPDO/output byte 3
//     MianTask Outputs/G_IO.arIOLinkRx_Place2[5]/OutputByte[0] <-> Module 6 (IOL_4/4_I/O-Bytes)/RxPDO/output byte 0
//     MianTask Outputs/G_IO.arIOLinkRx_Place2[5]/OutputByte[1] <-> Module 6 (IOL_4/4_I/O-Bytes)/RxPDO/output byte 1
//     MianTask Outputs/G_IO.arIOLinkRx_Place2[5]/OutputByte[2] <-> Module 6 (IOL_4/4_I/O-Bytes)/RxPDO/output byte 2
//     MianTask Outputs/G_IO.arIOLinkRx_Place2[5]/OutputByte[3] <-> Module 6 (IOL_4/4_I/O-Bytes)/RxPDO/output byte 3
//     MianTask Outputs/G_IO.arIOLinkRx_Place2[6]/OutputByte[0] <-> Module 7 (IOL_4/4_I/O-Bytes)/RxPDO/output byte 0
//     MianTask Outputs/G_IO.arIOLinkRx_Place2[6]/OutputByte[1] <-> Module 7 (IOL_4/4_I/O-Bytes)/RxPDO/output byte 1
//     MianTask Outputs/G_IO.arIOLinkRx_Place2[6]/OutputByte[2] <-> Module 7 (IOL_4/4_I/O-Bytes)/RxPDO/output byte 2
//     MianTask Outputs/G_IO.arIOLinkRx_Place2[6]/OutputByte[3] <-> Module 7 (IOL_4/4_I/O-Bytes)/RxPDO/output byte 3
//     MianTask Outputs/G_IO.arIOLinkRx_Place2[7]/OutputByte[0] <-> Module 8 (IOL_4/4_I/O-Bytes)/RxPDO/output byte 0
//     MianTask Outputs/G_IO.arIOLinkRx_Place2[7]/OutputByte[1] <-> Module 8 (IOL_4/4_I/O-Bytes)/RxPDO/output byte 1
//     MianTask Outputs/G_IO.arIOLinkRx_Place2[7]/OutputByte[2] <-> Module 8 (IOL_4/4_I/O-Bytes)/RxPDO/output byte 2
//     MianTask Outputs/G_IO.arIOLinkRx_Place2[7]/OutputByte[3] <-> Module 8 (IOL_4/4_I/O-Bytes)/RxPDO/output byte 3
//   Rohlik_Expansion/Rohlik_Expansion Instance <-> Place2/Term 36 (EK1100)/DI6
//     MianTask Inputs/G_IO.arDI[6]/Ch[{0..15}] <-> Channel {1..16}/Input  (16 links)
//   Rohlik_Expansion/Rohlik_Expansion Instance <-> Place2/Term 36 (EK1100)/DI7
//     MianTask Inputs/G_IO.arDI[7]/Ch[{0..15}] <-> Channel {1..16}/Input  (16 links)
//   Rohlik_Expansion/Rohlik_Expansion Instance <-> Place2/Term 36 (EK1100)/DO5
//     MianTask Outputs/G_IO.arDO[5]/Ch[{0..15}] <-> Channel {1..16}/Output  (16 links)
//   Rohlik_Expansion/Rohlik_Expansion Instance <-> Place2/Term 36 (EK1100)/DO7
//     MianTask Outputs/G_IO.arDO[7]/Ch[{0..15}] <-> Channel {1..16}/Output  (16 links)
//   Rohlik_Expansion/Rohlik_Expansion Instance <-> autoStore1/Term 56 (EK1100)/DI20
//     MianTask Inputs/G_IO.arDI[20]/Ch[{0..15}] <-> Channel {1..16}/Input  (16 links)
//   Rohlik_Expansion/Rohlik_Expansion Instance <-> autoStore2/Term 70 (EK1100)/DI21
//     MianTask Inputs/G_IO.arDI[21]/Ch[{0..15}] <-> Channel {1..16}/Input  (16 links)
//   Rohlik_Expansion/Rohlik_Expansion Instance <-> NC-Task 1 SAF/Axes/autostore1_lift
//     MianTask Inputs/GVL.fb_autoStore1.AxisRef_lift.NcToPlc <-> Outputs/ToPlc
//     MianTask Outputs/GVL.fb_autoStore1.AxisRef_lift.PlcToNc <-> Inputs/FromPlc
//   Rohlik_Expansion/Rohlik_Expansion Instance <-> NC-Task 1 SAF/Axes/autostore1_transfer
//     MianTask Inputs/GVL.fb_autoStore1.AxisRef_transfer.NcToPlc <-> Outputs/ToPlc
//     MianTask Outputs/GVL.fb_autoStore1.AxisRef_transfer.PlcToNc <-> Inputs/FromPlc
//   Rohlik_Expansion/Rohlik_Expansion Instance <-> NC-Task 1 SAF/Axes/autostore2_lift
//     MianTask Inputs/GVL.fb_autoStore2.AxisRef_lift.NcToPlc <-> Outputs/ToPlc
//     MianTask Outputs/GVL.fb_autoStore2.AxisRef_lift.PlcToNc <-> Inputs/FromPlc
//   Rohlik_Expansion/Rohlik_Expansion Instance <-> NC-Task 1 SAF/Axes/autostore2_transfer
//     MianTask Inputs/GVL.fb_autoStore2.AxisRef_transfer.NcToPlc <-> Outputs/ToPlc
//     MianTask Outputs/GVL.fb_autoStore2.AxisRef_transfer.PlcToNc <-> Inputs/FromPlc
//   Rohlik_Expansion/Rohlik_Expansion Instance <-> NC-Task 1 SAF/Axes/lift_motor
//     MianTask Inputs/GVL.fb_loading.AxisRef.NcToPlc <-> Outputs/ToPlc
//     MianTask Inputs/GVL.fb_loading.st_mcAxis.rActTorque <-> Outputs/ToPlc/ActTorque
//     MianTask Outputs/GVL.fb_loading.AxisRef.PlcToNc <-> Inputs/FromPlc
//   Rohlik_Expansion/Rohlik_Expansion Instance <-> NC-Task 1 SAF/Axes/working1_lift_motor
//     MianTask Inputs/GVL.fb_working1.AxisRef_lift.NcToPlc <-> Outputs/ToPlc
//     MianTask Inputs/GVL.fb_working1.st_mcAxis_lift.rActTorque <-> Outputs/ToPlc/ActTorque
//     MianTask Outputs/GVL.fb_working1.AxisRef_lift.PlcToNc <-> Inputs/FromPlc
//   Rohlik_Expansion/Rohlik_Expansion Instance <-> NC-Task 1 SAF/Axes/working1_open_bag
//     MianTask Inputs/GVL.fb_working1.AxisRef_bag.NcToPlc <-> Outputs/ToPlc
//     MianTask Inputs/GVL.fb_working1.st_mcAxis_bag.rActTorque <-> Outputs/ToPlc/ActTorque
//     MianTask Outputs/GVL.fb_working1.AxisRef_bag.PlcToNc <-> Inputs/FromPlc
//   Rohlik_Expansion/Rohlik_Expansion Instance <-> NC-Task 1 SAF/Axes/working2_lift_motor
//     MianTask Inputs/GVL.fb_working2.AxisRef_lift.NcToPlc <-> Outputs/ToPlc
//     MianTask Inputs/GVL.fb_working2.st_mcAxis_lift.rActTorque <-> Outputs/ToPlc/ActTorque
//     MianTask Outputs/GVL.fb_working2.AxisRef_lift.PlcToNc <-> Inputs/FromPlc
//   Rohlik_Expansion/Rohlik_Expansion Instance <-> NC-Task 1 SAF/Axes/working2_open_bag
//     MianTask Inputs/GVL.fb_working2.AxisRef_bag.NcToPlc <-> Outputs/ToPlc
//     MianTask Inputs/GVL.fb_working2.st_mcAxis_bag.rActTorque <-> Outputs/ToPlc/ActTorque
//     MianTask Outputs/GVL.fb_working2.AxisRef_bag.PlcToNc <-> Inputs/FromPlc

// ---- Ads/AutostoreStatus.TcDUT
{attribute 'qualified_only'}
{attribute 'strict'}
TYPE AutostoreStatus :
(
	UNKNOWN := 0,
	EXCHANGING	:=1,
	READY	:=2
);
END_TYPE

// ---- Mian/DUTs/E_WorkingStates.TcDUT
{attribute 'qualified_only'}
{attribute 'strict'}
TYPE E_WorkingStates ://can't divide into 2 states for load and unload,for sometimes if not unload,then call load,can cause accident
(
	IDLE := 0,
	INIT,
	CHECK,
	WAIT_NEW_TOTE,
	LOADING,
	WAIT_FINISHED,
	TOTE_LOAD,
	TOTE_UNLOAD,
	BAG_OPEN,
	BAG_OPEN_DETECTION,
	BAG_CLOSE_STEP_0,
	BAG_CLOSE_STEP_1,
	BAG_CLOSE,
	BAG_OPEN_INIT,
	TOTE_LIFT_UP,
	TOTE_LIFT_DOWN,
	BAG_OPEN_UP,
	WAIT_ROBORT_IN_SAFE_PLACE,
	BAG_OPEN_DOWN,
	TOTE_OUT,
	WAIT_1,
	
	WAIT_LOGTECH_OUTBOUND,
	TOTE_STATUS_DETECTION,
	
	NOTIFY_LOADING_OUTBOUND,
	
	AGING_STATE_0,
	AGING_STATE_1,

	WAIT,
	
	WAIT_UNLOADING,
	WAIT_SENSOR_ON,
	WAIT_SENSOR_OFF,
	WAIT_PREINBOUND_SENSOR_ON,
	WAIT_PREINBOUND_SENSOR_OFF,	
	WAIT_INBOUND_SENSOR_ON,
	WAIT_INBOUND_SENSOR_OFF,
	WAIT_LOAD_SENSOR_ON,
	WAIT_LOAD_SENSOR_OFF,
	WAIT_RECEIVE_TOTE_FINISHED,
	WAIT_TOTE_DETECTION_ON,
	WAIT_TOTE_DETECTION_OFF,
	DONE,
	ERROR
	
);
END_TYPE

// ---- GVLs/GVL_SAFETY.TcGVL
//{attribute 'qualified_only'}
VAR_GLOBAL
    	                                        	                                         
SO0_0              AT%I*  :BOOL           ;   //Robot1_EES急停         
SO0_1              AT%I*  :BOOL           ;   //Robot1_EAS安全门        
SO0_2              AT%I*  :BOOL           ;   //Robot2_EES急停  	                    
SO0_3              AT%I*  :BOOL           ;   //Robot2_EAS安全门  	    
                  
SO1_0              AT%I*  :BOOL           ;   //liftServo_STO1    升降伺服STO1
SO1_1              AT%I*  :BOOL           ;   //liftServo_STO2    升降伺服STO1
SO1_2              AT%I*  :BOOL           ;   //rollerBelt_Power  滚筒皮带电源STO控制	                    
SO1_3              AT%I*  :BOOL           ;   //NA
	                    
SO2_0              AT%I*  :BOOL           ;   //Place1_Servo_STO1 分拣1伺服STO1     
SO2_1              AT%I*  :BOOL           ;   //Place1_Servo_STO2 分拣1伺服STO2
SO2_2              AT%I*  :BOOL           ;   //rollerBelt_Power  滚筒皮带电源STO控制	
SO2_3              AT%I*  :BOOL           ;   //NA	
                    
SO3_0              AT%I*  :BOOL           ;   //Place2_Servo_STO1 分拣2伺服STO1    
SO3_1              AT%I*  :BOOL           ;   //Place_Servo_STO2  分拣2伺服STO2          
SO3_2              AT%I*  :BOOL           ;   //rollerBelt_Power  滚筒皮带电源STO控制
SO3_3              AT%I*  :BOOL           ;   //NA	       

SO4_0              AT%I*  :BOOL           ;   //Place2_Servo_STO1 分拣2伺服STO1    
SO4_1              AT%I*  :BOOL           ;   //Place_Servo_STO2  分拣2伺服STO2          
SO4_2              AT%I*  :BOOL           ;   //rollerBelt_Power  滚筒皮带电源STO控制
SO4_3              AT%I*  :BOOL           ;   //NA	                                                       
	                                        	 

b_FBerror					AT %I*	: BOOL;//安全功能块错误
b_ComError					AT %I*	: BOOL;//安全端口错误
	 
b_GroupRun					AT %Q*  : BOOL :=1;   //安全模块运行
b_ErrorAck					AT %Q*  : BOOL;     //安全模块错误确认
b_EStopRestart 				AT %Q* 	: BOOL;	//安全模块复位 	
bSafetyRestart_left			AT %Q* 	: BOOL; 
bSafetyRestart_right		AT %Q* 	: BOOL;
bSafetyReset_airDump	 	AT %Q* 	: BOOL;

bLeftDoorUnlock_Request 	AT %Q* : BOOL;	//TRUE:UNLOCK 	 
bRightDoorUnlock_Request 	AT %Q* : BOOL;	//TRUE:UNLOCK 


robots_ees_edm  			AT %Q* : BOOL ;

Robot1_EES_EDM  			AT %Q* : BOOL;
Robot2_EES_EDM  			AT %Q* : BOOL;
Robot1_EAS_EDM  			AT %Q* : BOOL;
Robot2_EAS_EDM  			AT %Q* : BOOL;
Lift_STO_EDM           		AT %Q* : BOOL;
Place1_STO_EDM         		AT %Q* : BOOL; 
Place2_STO_EDM        		AT %Q* : BOOL; 

robot1_STO_EES				AT %I* : BOOL;
robot1_STO_EAS				AT %I* : BOOL;	
robot2_STO_EES				AT %I* : BOOL;
robot2_STO_EAS				AT %I* : BOOL;
Lift_STO  		        	AT %I* : BOOL; 
Place1_STO	         		AT %I* : BOOL;
Place2_STO	        		AT %I* : BOOL; 
bAirDump1					AT %I* : BOOL; 
bAirDump2					AT %I* : BOOL; 
bAirDump1_feedback			AT %I* : BOOL; 
bAirDump2_feedback			AT %I* : BOOL; 



               
 END_VAR

// ---- Ads/FB_AirPressure_Subsystem.TcPOU
FUNCTION_BLOCK FB_AirPressure_Subsystem EXTENDS FB_Generic
VAR_INPUT

	 pPackTags		: POINTER TO ST_PackMLv30;
END_VAR
VAR_OUTPUT
END_VAR

VAR
ton1	: TON;
iCase	 : INT;
iAng_airPress	: INT;
iAng_airFlow		: INT;
air_pressure_status AT%Q* : AirPressureStatus; (* Current Air pressure status *)
air_pressure AT%Q*: REAL; (* Current air pressure value, MPa *)
air_flow AT%Q*: REAL; (* Current air flow value, L/min *)

rCurrent_flow	: REAL;
current_air_flow	: REAL; //unit: L/min
rTrig_error	:ARRAY[1..20] OF R_TRIG;
xError	: BOOL;
bAirDump_feedback	: BOOL;
END_VAR

VAR CONSTANT
	air_pressure_threshold_error AT%Q*: REAL:=0.4;//0.4*100 setting in PLC   (* Constant threshold of ERROR state for air pressure *)
	air_pressure_threshold_warning AT%Q*: REAL:=0.5;//0.5*100 setting in PLC (* Constant threshold of WARNING state for air pressure *)
    air_pressure_threshold_overtop AT%Q*: REAL:=1;//1*100 setting in PLC (* Constant threshold of OVERTOP state for air pressure *)
	
	rMin_voltage_flow	: REAL	:= 1.064;
	rMax_voltage_flow	: REAL	:= 5;
	rMaxFlow_L_per_minute		: REAL	:= 2000;
END_VAR

SUPER^();
IF sInstanceName='air_pressure1' THEN
	iAng_airPress	:=GVL.iAng_airPress_left;
	iAng_airFlow		:= GVL.iAng_AirFlow_left;	
	bAirDump_feedback			:= GVL_SAFETY.bAirDump1_feedback;
END_IF
IF sInstanceName='air_pressure2' THEN
	iAng_airPress	:=GVL.iAng_airPress_right;
	iAng_airFlow		:= GVL.iAng_AirFlow_right;
	bAirDump_feedback			:= GVL_SAFETY.bAirDump2_feedback;	
END_IF
xError	:= air_pressure_status=AirPressureStatus.ERROR OR bAirDump_feedback ;
///////////////////air_pressure//////////////////////////////
air_pressure	:= INT_TO_REAL(DINT_TO_INT(iAng_airPress*100/16#8000))/100;
IF air_pressure<air_pressure_threshold_error THEN
	air_pressure_status	:= AirPressureStatus.ERROR;
ELSIF air_pressure<air_pressure_threshold_warning THEN
	air_pressure_status	:= AirPressureStatus.WARNING;
ELSIF air_pressure<air_pressure_threshold_overtop THEN
	air_pressure_status	:= AirPressureStatus.HEALTH;
ELSE
	air_pressure_status	:= AirPressureStatus.OVERTOP;
END_IF
		
///////////////////air_flow//////////////////////////////
rCurrent_flow	:= INT_TO_REAL(iAng_airFlow*10)/16#8000;
IF rCurrent_flow>=1 THEN
	current_air_flow	:= rMaxFlow_L_per_minute*(rCurrent_flow-rMin_voltage_flow)/(rMax_voltage_flow-rMin_voltage_flow);
ELSE
	current_air_flow	:= 0;
END_IF		

air_flow:=REAL_TO_INT(current_air_flow);






rTrig_error[1](CLK:=air_pressure_status=AirPressureStatus.ERROR AND pPackTags^.Status.StateCurrent<>E_PMLState.ePMLState_Clearing);
IF pPackTags^.Status.StateCurrent<>E_PMLState.ePMLState_Resetting THEN
	FOR i:=1 TO 20 DO
		IF rTrig_error[i].Q THEN
			THIS^.packTags.Admin.Alarm[i].ID	:= i;
			CASE i OF
				1:
					THIS^.packTags.Admin.Alarm[1].Message	:= GenerateErrorMsg(errorType:='A',iState := i,errorMsg:='Air pressure is low');
			END_CASE
			THIS^.pml_adminAlarm.M_SetAlarm(stAdmin:=pPackTags^.Admin,stAlarm := THIS^.packTags.Admin.Alarm[i]);
		END_IF
	END_FOR
END_IF

END_FUNCTION_BLOCK

// ---- Ads/FB_HeartBeat_Subsystem.TcPOU
FUNCTION_BLOCK FB_HeartBeat_Subsystem EXTENDS FB_Generic
VAR_INPUT
	
END_VAR
VAR_OUTPUT
	heart_timeout_Alarm:BOOL;
END_VAR
VAR
	bReset_ads_heart_beat	: HeartbeatParams;
	bReset_ads_heart_beatTemp	: HeartbeatParams;
	heart_timeout:TON;
	AA: INT;
	rtrig_abort	: R_TRIG;
END_VAR

heart_timeout(PT:=T#3S);

IF bReset_ads_heart_beat.current_time_ms=bReset_ads_heart_beatTemp.current_time_ms THEN
	heart_timeout.IN	:=TRUE;
ELSE
	heart_timeout.IN	:=FALSE;
	heart_timeout_Alarm:=FALSE;
	bReset_ads_heart_beatTemp.current_time_ms	:= bReset_ads_heart_beat.current_time_ms;	
END_IF

IF heart_timeout.Q  THEN
	heart_timeout.IN:=FALSE;
	heart_timeout_Alarm:=TRUE;
	
END_IF

rtrig_abort(CLK	:= heart_timeout_Alarm);
IF rtrig_abort.Q THEN
	IF sInstanceName='heartBeat_1' THEN
		subData.Topic	:= E_Topics.WORKING1_ABORT_INBOUND;
		GVL.PubSubService.Publish(topic:=E_Topics.WORKING1_ABORT_INBOUND,data:= subData);
		subData.Topic	:= E_Topics.WORKING1_ABORT_OUTBOUND;
		GVL.PubSubService.Publish(topic:=E_Topics.WORKING1_ABORT_OUTBOUND,data:= subData);	
	END_IF	
	IF sInstanceName='heartBeat_2' THEN
		subData.Topic	:= E_Topics.WORKING2_ABORT_INBOUND;
		GVL.PubSubService.Publish(topic:=E_Topics.WORKING2_ABORT_INBOUND,data:= subData);	
		subData.Topic	:= E_Topics.WORKING2_ABORT_OUTBOUND;
		GVL.PubSubService.Publish(topic:=E_Topics.WORKING2_ABORT_OUTBOUND,data:= subData);		
	END_IF		
END_IF

{attribute 'TcRpcEnable'}
METHOD heartbeat : UDINT
VAR_INPUT
	heartbeat_params : HeartbeatParams;	
END_VAR
heartbeat	:= 1; 
bReset_ads_heart_beat	:= heartbeat_params;
heartbeat	:= MethodCallReturnValue.ACCEPTED;

AA:=AA+1;
END_METHOD

END_FUNCTION_BLOCK

// ---- Ads/FB_Safety_Subsystem.TcPOU
FUNCTION_BLOCK FB_Safety_Subsystem EXTENDS FB_Generic
VAR_INPUT
	pHeartBeat		: POINTER TO FB_HeartBeat_Subsystem;
	pSafety_door	: POINTER TO ST_safetyDoor;
	pPackTags		: POINTER TO ST_PackMLv30;
	pMachine		: POINTER TO FB_Machine;
END_VAR
VAR_IN_OUT
	
END_VAR
VAR_OUTPUT
	
END_VAR
VAR
	button_array AT%Q* : ARRAY [0..99] OF ButtonStatus; (* Array of 100 elements for ButtonStatus, button reset, button unlock *)
	estop_array AT%Q* : ARRAY [0..99] OF EStopStatus; (* Array of 100 elements for EStopStatus *)
	safety_door_array AT%Q*: ARRAY [0..99] OF SafetyDoorStatus; (* Array of 100 elements for SafetyDoorStatus *)
	light_curtain_array AT%Q*: ARRAY [0..999] OF LightCurtainStatus; (* Array of 1000 elements for LightCurtainStatus *)
	sensor_array  AT%Q*: ARRAY [0..999] OF SensorStatus; (* Array of 1000 elements for SensorStatus *)
	estop_status AT%Q*: GeneralStatus;
	gates_status AT%Q*: GeneralStatus;
	safety_status AT%Q*: GeneralStatus;

	SI_0	: UINT;
	SI_1	: UINT;
	GI_0 	: UINT;
	GI_1 	: UINT;
	
	
	station_mode	: StationMode;//APP status
	iStationMode	: UINT;
	iState: INT;
	bEstop_detection	: BOOL;	
	

	eStates					:	E_SafetyStates	:=	E_SafetyStates.IDLE;
	eStateTemp				:	E_SafetyStates	:=	E_SafetyStates.IDLE;

	errorMessage	: STRING;
	xError	: BOOL;
	xEstop	: BOOL;
	xError_working	: BOOL;
	xEstop_behavior	: BOOL;
	
	xError_loading	: BOOL;
	eStates_safetyDoor	: E_SAFETYDOOR	:= E_SAFETYDOOR.IDLE;
	bReset_safetyDoor	: BOOL;
	
	
	
	GPWM	: FB_GPWM;
	GPWM_1s	: FB_GPWM;
	tonSaftyDelay: TON;
	b_EStopRestarting  : BOOL;
	T_EStopRestart : TON;
//////////////////////SAFETY hardware config///////////////	
	mcp_estop_left				: FB_DigitalInput;
	safetyDoor_left				: BOOL;
	
	mcp_estop_right				: FB_DigitalInput;
	safetyDoor_right			: BOOL;
	door_closed					: BOOL;
	bRobot1_eStop				: BOOL;
	bRobot2_eStop				: BOOL;

	lift_station_detection		: BOOL;
	
	lift_door_left				: FB_DigitalInput;
	lift_door_right				: FB_DigitalInput;
	
	robot1_EES					: BOOL;
	robot1_EAS					: BOOL;
	
	robot2_EES					: BOOL;
	robot2_EAS					: BOOL;
	buffer_safety				: BOOL;
	loading_safety				: BOOL;
	working_safety				: BOOL;
	baffle_sensor_1				: BOOL;
	baffle_sensor_2				: BOOL;
	
	LiftStoEDM					: BOOL;
	Place1StoEDM				: BOOL;
	Place2StoEDM				: BOOL;  

	
	safety_door_unlock_en		: BOOL;
	bStop_button_unlock		: BOOL;//for not receive cmd from tote_subsystem
	

	
	
	refMachineCmd	: REFERENCE TO E_PMLCommand;
	lift_safetyDoor_left: BOOL;
	lift_safetyDoor_right: BOOL;
	

	
	ton_waitDoorLocked	: TON;
	
	pml_command	: E_PMLCommand;
	
	bDoorUnlockRequest	: BOOL;
	fTrig_error	:ARRAY[1..20] OF F_TRIG;
	
	resetting	: BOOL;//while in resetting,can not unlock the door
	
	ESLE: INT;
END_VAR

SUPER^();
M_mapping();
M_safetyDoor();


IF sInstanceName='safety_1' THEN
	IF pMachine^.eState=ePMLState_Aborted THEN 
		IF xEstop AND pSafety_door^.door_locked AND (GVL.fb_mcp_2.st_safety_door.door_locked OR lift_door_right.Q) THEN
			pSafety_door^.lamp_reset	:= GPWM_1s.q_xOut;
		ELSE
			pSafety_door^.lamp_reset	:= TRUE;
		END_IF	
	ELSE
		pSafety_door^.lamp_reset	:= FALSE;
	END_IF
END_IF
IF sInstanceName='safety_2' THEN
	IF pMachine^.eState=ePMLState_Aborted THEN
		IF xEstop AND pSafety_door^.door_locked AND (GVL.fb_mcp_1.st_safety_door.door_locked OR lift_door_left.Q) THEN
			pSafety_door^.lamp_reset	:= GPWM_1s.q_xOut;
		ELSE
			pSafety_door^.lamp_reset	:= TRUE;
		END_IF
	ELSE
		pSafety_door^.lamp_reset	:= FALSE;
	END_IF	
END_IF

xEstop	:= bRobot1_eStop AND bRobot2_eStop AND mcp_estop_left.Q AND mcp_estop_right.Q AND lift_station_detection AND baffle_sensor_1 AND baffle_sensor_2;
xEstop_behavior	:= NOT(GVL_SAFETY.robot1_STO_EES AND GVL_SAFETY.robot2_STO_EES AND GVL_SAFETY.Lift_STO);
IF sInstanceName='safety_1' THEN
		xError	:=NOT(GVL_SAFETY.robot1_STO_EES AND GVL_SAFETY.Lift_STO AND GVL_SAFETY.Place1_STO AND GVL_SAFETY.robot1_STO_EAS); 
		GVL_SAFETY.bLeftDoorUnlock_Request	:= pSafety_door^.door_lock;		
		IF robot1_EES THEN 
			IF robot1_EAS THEN
				safety_status := GeneralStatus.READY ;
			ELSE
				safety_status := GeneralStatus.NOT_READY ;
			END_IF
		ELSE
			safety_status := GeneralStatus.ERROR; 
		END_IF
END_IF
IF sInstanceName='safety_2' THEN
	xError	:=NOT(GVL_SAFETY.robot2_STO_EES AND GVL_SAFETY.Lift_STO AND GVL_SAFETY.Place2_STO AND GVL_SAFETY.robot2_STO_EAS);
	GVL_SAFETY.bRightDoorUnlock_Request	:= pSafety_door^.door_lock;
	IF robot2_EES THEN 
		IF robot2_EAS THEN
			safety_status := GeneralStatus.READY ;
		ELSE
			safety_status := GeneralStatus.NOT_READY ;
		END_IF
	ELSE
		safety_status := GeneralStatus.ERROR; 
	END_IF		
END_IF

//安全Safety报警 确认 复位
tonSaftyDelay(IN:= NOT tonSaftyDelay.Q ,PT:=T#1S);
b_ErrorAck := tonSaftyDelay.Q;


GPWM(i_xEnable:=TRUE,i_udiTime:=10,i_udiCycle:=20);
GPWM_1s(i_xEnable:=TRUE,i_udiTime:=500,i_udiCycle:=1000);

 



////////////////////////////////////////////////safety error/////////////////////////////////////////////////// 
IF wcState_mcp=0 AND wcState_lift=0 AND wcState_place1=0 AND wcState_place2=0 THEN
	fTrig_error[1](CLK:=mcp_estop_left.Q OR pMachine^.eState = ePMLState_Clearing);
	fTrig_error[2](CLK:=mcp_estop_right.Q OR pMachine^.eState = ePMLState_Clearing);
	fTrig_error[3](CLK:=bRobot1_eStop OR pMachine^.eState = ePMLState_Clearing);
	fTrig_error[4](CLK:=bRobot2_eStop OR pMachine^.eState = ePMLState_Clearing);
	fTrig_error[5](CLK:=lift_station_detection OR pMachine^.eState = ePMLState_Clearing);
	fTrig_error[6](CLK:=baffle_sensor_1 OR pMachine^.eState = ePMLState_Clearing);
	fTrig_error[7](CLK:= baffle_sensor_2 OR pMachine^.eState = ePMLState_Clearing);
	IF sInstanceName='safety_1' THEN
		fTrig_error[8](CLK:=safetyDoor_left OR pMachine^.eState = ePMLState_Clearing);
	END_IF
	IF sInstanceName='safety_2' THEN
		fTrig_error[8](CLK:=safetyDoor_right OR pMachine^.eState = ePMLState_Clearing);
	END_IF
END_IF
fTrig_error[9](CLK:= wcState_mcp=0 OR pMachine^.eState = ePMLState_Clearing);
fTrig_error[10](CLK:= wcState_lift=0 OR pMachine^.eState = ePMLState_Clearing);
fTrig_error[11](CLK:= wcState_place1=0 OR pMachine^.eState = ePMLState_Clearing);
fTrig_error[12](CLK:= wcState_place2=0 OR pMachine^.eState = ePMLState_Clearing);
IF pPackTags^.Status.StateCurrent<>E_PMLState.ePMLState_Resetting THEN
	FOR i:=1 TO 20 DO
		IF fTrig_error[i].Q THEN
			THIS^.packTags.Admin.Alarm[i].ID	:= i;
			CASE i OF
				1:
					THIS^.packTags.Admin.Alarm[1].Message	:= GenerateErrorMsg(errorType:='S',iState := i,errorMsg:='estop on left door is pressed');
				2:
					THIS^.packTags.Admin.Alarm[2].Message	:= GenerateErrorMsg(errorType:='S',iState := i,errorMsg:='estop on right door is pressed');
				3:
					THIS^.packTags.Admin.Alarm[3].Message	:= GenerateErrorMsg(errorType:='S',iState := i,errorMsg:='estop on robot1 teachpannel is pressed');
				4:
					THIS^.packTags.Admin.Alarm[4].Message	:= GenerateErrorMsg(errorType:='S',iState := i,errorMsg:='estop on robot2 teachpannel is pressed');
				5:
					THIS^.packTags.Admin.Alarm[5].Message	:= GenerateErrorMsg(errorType:='S',iState := i,errorMsg:='switch detecting lift module is not detected');
				6:
					THIS^.packTags.Admin.Alarm[6].Message	:= GenerateErrorMsg(errorType:='S',iState := i,errorMsg:='up baffle is not detected');	
				7:
					THIS^.packTags.Admin.Alarm[7].Message	:= GenerateErrorMsg(errorType:='S',iState := i,errorMsg:='down baffle is not detected');	
				8:
					THIS^.packTags.Admin.Alarm[8].Message	:= GenerateErrorMsg(errorType:='S',iState := i,errorMsg:='gate is unlocked');	
				9:
					THIS^.packTags.Admin.Alarm[9].Message	:= GenerateErrorMsg(errorType:='S',iState := i,errorMsg:='MCP EtherCAT bus is in state ERROR');	
				10:
					THIS^.packTags.Admin.Alarm[10].Message	:= GenerateErrorMsg(errorType:='S',iState := i,errorMsg:='Lift module EtherCAT bus is in state ERROR');	
				11:
					THIS^.packTags.Admin.Alarm[11].Message	:= GenerateErrorMsg(errorType:='S',iState := i,errorMsg:='Place1 module EtherCAT bus is in state ERROR');	
				12:
					THIS^.packTags.Admin.Alarm[12].Message	:= GenerateErrorMsg(errorType:='S',iState := i,errorMsg:='Place2 module EtherCAT bus is in state ERROR');	

			END_CASE
			THIS^.pml_adminAlarm.M_SetAlarm(stAdmin:=pPackTags^.Admin,stAlarm := THIS^.packTags.Admin.Alarm[i]);
		END_IF
	END_FOR
END_IF

PROPERTY _stationMode : StationMode
GET
_stationMode	:= station_mode;
END_GET
SET
station_mode	:= _stationMode;
END_SET
END_PROPERTY

METHOD M_mapping : BOOL
VAR_INPUT
END_VAR

VAR

	
END_VAR


mcp_estop_left(D:= G_IO.arSI[0].Ch[1] AND G_IO.arSI[0].Ch[2],on_ms:=100,off_ms:=50);//while trig door lock and unlock,it will trig the input randomly	
safetyDoor_left				:= G_IO.arSI[0].Ch[3] AND G_IO.arSI[0].Ch[4];
mcp_estop_right(D:= G_IO.arSI[1].Ch[1] AND G_IO.arSI[1].Ch[2],on_ms:=100,off_ms:=50);//while trig door lock and unlock,it will trig the input randomly	
safetyDoor_right			:= G_IO.arSI[1].Ch[3] AND G_IO.arSI[1].Ch[4];
IF sInstanceName='safety_1' THEN
	door_closed					:= G_IO.arSI[2].Ch[3];
	
END_IF
IF sInstanceName='safety_2' THEN
	door_closed					:= G_IO.arSI[2].Ch[4];
END_IF
bRobot1_eStop				:= G_IO.arSI[3].Ch[1] AND G_IO.arSI[3].Ch[2];
bRobot2_eStop				:= G_IO.arSI[3].Ch[3] AND G_IO.arSI[3].Ch[4];

lift_station_detection		:= G_IO.arSI[4].Ch[3] AND G_IO.arSI[4].Ch[4];
lift_door_left(D:= G_IO.arSI[5].Ch[1] AND G_IO.arSI[5].Ch[2],on_ms:=500,off_ms:=80);
lift_door_right(D:= G_IO.arSI[5].Ch[3] AND G_IO.arSI[5].Ch[4],on_ms:=500,off_ms:=80);
baffle_sensor_1				:= G_IO.arSI[6].Ch[1] AND G_IO.arSI[6].Ch[2];
baffle_sensor_2				:= G_IO.arSI[6].Ch[3] AND G_IO.arSI[6].Ch[4];
bAirDump1_feedback			:= arDI[1].Ch[0] AND arDI[1].Ch[1];
bAirDump2_feedback			:= arDI[1].Ch[8] AND arDI[1].Ch[9];
	
robot1_EES					:= GVL_SAFETY.robot1_STO_EES;
robot1_EAS					:= GVL_SAFETY.robot1_STO_EAS;
robot2_EES					:= GVL_SAFETY.robot2_STO_EES;
robot2_EAS					:= GVL_SAFETY.robot2_STO_EAS;
LiftStoEDM					:= GVL_SAFETY.Lift_STO_EDM;
Place1StoEDM				:= GVL_SAFETY.Place1_STO_EDM;
Place2StoEDM				:= GVL_SAFETY.Place2_STO_EDM;                 
                    
                  
 //EDM config
// GVL_IOLink.robots_ees_edm  	:= TRUE;  
 GVL_SAFETY.Robot1_EES_EDM  	:= GVL.fb_mcp_1.EDM_EES;
 GVL_SAFETY.Robot2_EES_EDM  	:= GVL.fb_mcp_2.EDM_EES; 
 GVL_SAFETY.robot1_eas_edm  	:= GVL.fb_mcp_1.EDM_EAS;
 GVL_SAFETY.robot2_eas_edm  	:= GVL.fb_mcp_2.EDM_EAS;
// GVL_SAFETY.Lift_STO_EDM        := GVL.fb_loading.EDM_KM;
// GVL_SAFETY.Place1_STO_EDM      := GVL.fb_working1.EDM_KM;
// GVL_SAFETY.Place2_STO_EDM      := GVL.fb_working2.EDM_KM;	
	



/////////////////////////////////////////////Estop array//////////////////////////////////
IF mcp_estop_left.Q THEN
	estop_array[0]:=EStopStatus.DISENGAGED;
ELSE
	estop_array[0]:=EStopStatus.ENGAGED;	
END_IF
IF mcp_estop_right.Q THEN
	estop_array[1]:=EStopStatus.DISENGAGED;
ELSE
	estop_array[1]:=EStopStatus.ENGAGED;	
END_IF
IF bRobot1_eStop THEN
	estop_array[2]:=EStopStatus.DISENGAGED;
ELSE
	estop_array[2]:=EStopStatus.ENGAGED;	
END_IF
IF bRobot2_eStop THEN
	estop_array[3]:=EStopStatus.DISENGAGED;
ELSE
	estop_array[3]:=EStopStatus.ENGAGED;	
END_IF

/////////////////////////////////////////////button array//////////////////////////////////

IF pSafety_door^.button_reset THEN
	button_array[0]:=ButtonStatus.PRESSED;
ELSE
	button_array[0]:=ButtonStatus.RELEASED;	
END_IF
IF pSafety_door^.button_unlock THEN
	button_array[1]:=ButtonStatus.PRESSED;
ELSE
	button_array[1]:=ButtonStatus.RELEASED;	
END_IF
/////////////////////////////////////////////safety door array//////////////////////////////////
IF sInstanceName='safety_1' THEN
	IF safetyDoor_left THEN
		safety_door_array[0]:=SafetyDoorStatus.LOCKED;
	ELSE
		safety_door_array[0]:=SafetyDoorStatus.UNLOCKED;
	END_IF
END_IF
IF sInstanceName='safety_2' THEN
	IF safetyDoor_right THEN
		safety_door_array[0]:=SafetyDoorStatus.LOCKED;
	ELSE
		safety_door_array[0]:=SafetyDoorStatus.UNLOCKED;
	END_IF	
END_IF   
/////////////////////////////////////////////sensor array//////////////////////////////////
IF lift_station_detection THEN
	sensor_array[0]:=SensorStatus.SIGNAL;
ELSE
	sensor_array[0]:=SensorStatus.NO_SIGNAL;
END_IF
IF baffle_sensor_1 THEN
	sensor_array[1]:=SensorStatus.SIGNAL;
ELSE
	sensor_array[1]:=SensorStatus.NO_SIGNAL;
END_IF
IF baffle_sensor_2 THEN
	sensor_array[2]:=SensorStatus.SIGNAL;
ELSE
	sensor_array[2]:=SensorStatus.NO_SIGNAL;
END_IF
IF lift_door_left.Q THEN
	sensor_array[3]:=SensorStatus.SIGNAL;
ELSE
	sensor_array[3]:=SensorStatus.NO_SIGNAL;
END_IF

IF lift_door_right.Q THEN
	sensor_array[4]:=SensorStatus.SIGNAL;
ELSE
	sensor_array[4]:=SensorStatus.NO_SIGNAL;
END_IF
IF pSafety_door^.door_closed THEN
	sensor_array[5]:=SensorStatus.SIGNAL;
ELSE
	sensor_array[5]:=SensorStatus.NO_SIGNAL;
END_IF
//GI_0.0	:= GVL.fb_mcp.st_safety_door.button_reset;
//GI_0.1	:= GVL.fb_mcp.st_safety_door.button_unlock;
//GI_0.2	:= GVL.fb_mcp.st_safety_door.door_closed;

//SI_0.0	:= mcp_estop_left;
//SI_0.1	:= safetyDoor_left;
//SI_0.2	:= belt_estop;
//SI_0.3	:= lift_estop;
//SI_0.4	:= lift_station_detection;
END_METHOD

METHOD M_reset : BOOL
VAR_INPUT
	
END_VAR
M_reset	:= FALSE;
resetting	:= TRUE;
//xError	:= FALSE;//remove while safety is ready
//M_reset	:= TRUE;//remove while safety is ready
//RETURN;//remove while safety is ready
//check if all safety outputs
//////////////////////////////////////////////////////////timeout//////////////////////////////////////////
		ton_timeout();
		iStateTemp	:= eStateTemp;
		IF eStateTemp=eStates THEN
			ton_timeout.IN	:=TRUE;
		ELSE
			ton_timeout.IN	:=FALSE;
			eStateTemp	:= eStates;	
			M_Log(eLogType:=ServerityLevelType.INFO,sTextLog:='');
			IF ton_timeout.Q THEN
				RETURN;
			END_IF
		END_IF
		IF ton_timeout.Q THEN	
			ton_timeout.IN	:=FALSE;
			CASE eStates OF	
				E_SafetyStates.ERROR:	
					alarm_temp.Message	:= GenerateErrorMsg(errorType:='S',iState := iStateTemp,errorMsg:='in error state.');
				ELSE
					alarm_temp.Message	:= GenerateErrorMsg(errorType:='S',iState := iStateTemp,errorMsg:='time out');
			END_CASE
//////////////////////////////////////////////////////////states don't want to timeout and trig error//////////////////////////////////////////				
			IF  eStates<>E_SafetyStates.IDLE AND
				eStates<>E_SafetyStates.TRIG_RESET
			THEN
				eStates	:= E_SafetyStates.ERROR;
				IF sInstanceName='safety_1' THEN					
					THIS^.pml_adminAlarm.M_SetAlarm(stAdmin:=GVL.PackTags1.Admin,stAlarm:=THIS^.alarm_temp);
				END_IF			
				IF sInstanceName='safety_2' THEN
					THIS^.pml_adminAlarm.M_SetAlarm(stAdmin:=GVL.PackTags2.Admin,stAlarm:=THIS^.alarm_temp);
				END_IF					
			END_IF
		END_IF


CASE eStates OF
	E_SafetyStates.IDLE:
		pml_command	:= ePMLCommand_Undefined;
		xError	:= FALSE;
		ton_timeout.PT	:= T#1000MS;
		eStates	:= E_SafetyStates.CHECK_SAFETY_INPUTS;
	E_SafetyStates.CHECK_SAFETY_INPUTS:
		IF xEstop AND pSafety_door^.door_locked THEN
			eStates	:= E_SafetyStates.CHECK_OTHER_STATION;
		END_IF
	E_SafetyStates.CHECK_OTHER_STATION:
		IF sInstanceName='safety_1' THEN
			IF GVL.fb_mcp_2.st_safety_door.door_locked OR lift_door_right.Q THEN
				eStates	:= E_SafetyStates.TRIG_RESET;
			END_IF
		END_IF
		IF sInstanceName='safety_2' THEN
			IF GVL.fb_mcp_1.st_safety_door.door_locked OR lift_door_left.Q THEN
				eStates	:= E_SafetyStates.TRIG_RESET;
			END_IF
		END_IF
	E_SafetyStates.TRIG_RESET:
		ton_timeout.PT	:= T#300MS;
		b_EStopRestart	:= GPWM.q_xOut;
		IF sInstanceName='safety_1' THEN
			bSafetyRestart_left		:= GPWM.q_xOut;
		END_IF
		IF sInstanceName='safety_2' THEN	
			bSafetyRestart_right	:= GPWM.q_xOut;
		END_IF
		IF ton_timeout.Q THEN
			b_EStopRestart	:= FALSE;
			bSafetyRestart_left		:= FALSE;
			bSafetyRestart_right	:= FALSE;
			eStates	:= E_SafetyStates.CHECK_SAFETY_OUTPUT;
		END_IF		
	E_SafetyStates.CHECK_SAFETY_OUTPUT:	
		IF sInstanceName='safety_1' THEN
			IF Lift_STO AND Place1_STO THEN
				eStates	:= E_SafetyStates.LOCKDOOR_REQUEST;
			END_IF
		END_IF			
		IF sInstanceName='safety_2' THEN
			IF Lift_STO AND Place2_STO THEN
				eStates	:= E_SafetyStates.LOCKDOOR_REQUEST;		
			END_IF	
		END_IF
	E_SafetyStates.LOCKDOOR_REQUEST:
		ton_timeout.PT	:= T#3000MS;
		IF sInstanceName='safety_1' THEN
			IF GVL.fb_loading.M_LockRequest_1() THEN
				eStates	:= E_SafetyStates.DONE;
			END_IF			
		END_IF
		IF sInstanceName='safety_2' THEN
			IF GVL.fb_loading.M_LockRequest_2() THEN
				eStates	:= E_SafetyStates.DONE;
			END_IF			
		END_IF			
	E_SafetyStates.DONE:
		M_reset	:= TRUE;
		resetting	:= FALSE;
		eStates	:= E_SafetyStates.IDLE;
	E_SafetyStates.ERROR:	
		M_reset	:= TRUE;
		resetting	:= FALSE;
		xError	:= TRUE;
		eStates	:= E_SafetyStates.IDLE;

	
END_CASE
END_METHOD

(*
	button_lock:lock the gate and then control the related door of lift  
	button_unlock:	1)wait station stopped 
					2)control the related doors
					3)unlock the gate
	button_reset:	1)reset safety 
					2)control the related door of lift module
*)
METHOD M_safetyDoor : BOOL
VAR_INPUT
	
END_VAR

safety_door_unlock_en	:= (safety_status<>GeneralStatus.READY OR 
							(station_mode = StationMode.STOPPED OR 
							station_mode = StationMode.DISABLED OR
							station_mode = StationMode.INTERVENTION OR 
							pHeartBeat^.heart_timeout_Alarm)) AND
							(pMachine^.eState=ePMLState_Aborted OR 
							pMachine^.eState=ePMLState_Stopped OR	
							pMachine^.eState=ePMLState_Idle);

ton_waitDoorLocked(PT:=T#1000MS);
IF NOT xEstop THEN
	eStates_safetyDoor	:= E_SAFETYDOOR.UNLOCKING;	
END_IF			
CASE eStates_safetyDoor	OF
	E_SAFETYDOOR.IDLE:
		IF pSafety_door^.door_locked THEN
			eStates_safetyDoor	:= E_SAFETYDOOR.LOCKED;
		ELSE
			eStates_safetyDoor	:= E_SAFETYDOOR.UNLOCKED;
		END_IF
	E_SAFETYDOOR.LOCKED:
		pSafety_door^.lamp_lock	:=	FALSE;
		pSafety_door^.lamp_unlock	:= TRUE;//door lcoked,unlock lamp solid
		IF pSafety_door^.button_unlock AND NOT resetting THEN//while resetting,door can not be unlock,otherwise might trig safety
			bStop_button_unlock	:= TRUE;
			eStates_safetyDoor	:= E_SAFETYDOOR.WAIT_UNLOCK_EN;
		END_IF			
	E_SAFETYDOOR.REQUEST_LOCK:
	;
	E_SAFETYDOOR.SAFETY:
	;
	E_SAFETYDOOR.UNLOCKED:
		pSafety_door^.lamp_unlock	:= FALSE;
		IF pSafety_door^.door_closed THEN
			pSafety_door^.lamp_lock	:= GPWM_1s.q_xOut;//door closed,lock lamp blinking
			IF pSafety_door^.button_lock THEN
				bStop_button_unlock	:= FALSE;
				eStates_safetyDoor	:= E_SAFETYDOOR.WAIT_LOCKED;
			END_IF
		ELSE
			pSafety_door^.lamp_lock	:= TRUE;//door open,lock lamp solid
		END_IF
	E_SAFETYDOOR.WAIT_LOCKED:
		ton_waitDoorLocked.IN	:= TRUE;
		pSafety_door^.door_lock	:= FALSE;
		IF pSafety_door^.door_locked THEN
			ton_waitDoorLocked.IN	:= FALSE;
			eStates_safetyDoor	:= E_SAFETYDOOR.LOCKED;
	 	END_IF
		//if lock door failed,turn to unlock door and need to press the lock button to lock the door once more
		IF ton_waitDoorLocked.Q THEN
			ton_waitDoorLocked.IN	:= FALSE;
			eStates_safetyDoor	:= E_SAFETYDOOR.UNLOCKING;
		END_IF
		
	E_SAFETYDOOR.WATI_LODING_DOOR://wait the state of lift door
		pSafety_door^.lamp_unlock	:= GPWM_1s.q_xOut;//door unlocking,unlock lamp blinking
		IF sInstanceName='safety_1' THEN
			IF bAirDump1 AND NOT bAirDump1_feedback THEN//while gate is locked and its air is dumpped,means safety error must be accupped 
				IF GVL.fb_loading.M_unlockRequest(sInstanceName:=sInstanceName) THEN
					eStates_safetyDoor	:= E_SAFETYDOOR.UNLOCKING;
				END_IF
			ELSE
				eStates_safetyDoor	:= E_SAFETYDOOR.UNLOCKING;	
			END_IF		
		END_IF	
		IF sInstanceName='safety_2' THEN
			IF bAirDump2 AND NOT bAirDump2_feedback THEN//while gate is locked and its air is dumpped,means safety error must be accupped 
				IF GVL.fb_loading.M_unlockRequest(sInstanceName:=sInstanceName) THEN
					eStates_safetyDoor	:= E_SAFETYDOOR.UNLOCKING;
				END_IF
			ELSE
				eStates_safetyDoor	:= E_SAFETYDOOR.UNLOCKING;	
			END_IF			
		END_IF
	E_SAFETYDOOR.WAIT_UNLOCK_EN:
		IF pHeartBeat^.heart_timeout_Alarm OR (station_mode = StationMode.INTERVENTION AND pSafety_door^.button_unlock) THEN
			pml_command	:= ePMLCommand_Stop;
		END_IF
		
		pSafety_door^.lamp_unlock	:= GPWM_1s.q_xOut;//door unlocking,unlock lamp blinking
		IF safety_door_unlock_en THEN
			pml_command	:= ePMLCommand_Undefined;
			eStates_safetyDoor	:= E_SAFETYDOOR.WATI_LODING_DOOR;
		END_IF
	E_SAFETYDOOR.UNLOCKING:
		pml_command	:= ePMLCommand_Undefined;
		pSafety_door^.lamp_unlock	:= GPWM_1s.q_xOut;//door unlocking,unlock lamp blinking
		pSafety_door^.door_lock	:= TRUE;
		IF NOT pSafety_door^.door_locked THEN
			eStates_safetyDoor	:= E_SAFETYDOOR.UNLOCKED;
		END_IF
	
END_CASE
END_METHOD

METHOD ParseStateToString : STRING
VAR_INPUT
END_VAR
CASE THIS^.eStates OF
	E_SafetyStates.IDLE:
		ParseStateToString	:='IDLE';
	E_SafetyStates.CHECK_SAFETY_INPUTS:
		ParseStateToString	:='CHECK_SAFETY_INPUTS';
	E_SafetyStates.CHECK_DOOR_CLOSED:
		ParseStateToString	:='CHECK_DOOR_CLOSED';
	E_SafetyStates.CHECK_DOOR_LOCKED:
		ParseStateToString	:='CHECK_DOOR_LOCKED';
	E_SafetyStates.LOCKDOOR_REQUEST:
		ParseStateToString	:='LOCKDOOR_REQUEST';
	E_SafetyStates.CHECK_DOOR_OSSD:
		ParseStateToString	:='CHECK_DOOR_OSSD';
	E_SafetyStates.CHECK_SAFETY_OUTPUT:
		ParseStateToString	:='CHECK_SAFETY_OUTPUT';
	E_SafetyStates.DOOR_LOCK:
		ParseStateToString	:='DOOR_LOCK';
	E_SafetyStates.TRIG_RESET:
		ParseStateToString	:='TRIG_RESET';
	E_SafetyStates.CHECK_OTHER_STATION:
		ParseStateToString	:='CHECK_OTHER_STATION';
	E_SafetyStates.DONE:
		ParseStateToString	:='DONE';
	E_SafetyStates.ERROR:
		ParseStateToString	:='ERROR';
	ELSE
		ParseStateToString	:='UNKNOW STATE';
END_CASE
END_METHOD

{attribute 'TcRpcEnable'}
METHOD update_station_mode  : UDINT
VAR_INPUT
	update_station_mode_params	: UpdateStationModeParams;
END_VAR
update_station_mode	:= 1;
station_mode	:= update_station_mode_params.station_mode;
update_station_mode	:= 0;
END_METHOD

END_FUNCTION_BLOCK

// ---- Ads/FB_Tote_Subsystem.TcPOU
FUNCTION_BLOCK FB_Tote_Subsystem EXTENDS FB_Generic
VAR_INPUT
	
END_VAR
VAR_OUTPUT
END_VAR
VAR
	tote_status_array 	AT%Q*	: ARRAY [0..99] OF ToteStatus;
	
	status					: MachineStatus := MachineStatus.STOPPED;	
	current_air_pressure	: REAL;	
	machine_control_cmd	 	: MachineControlCommand;
	
	cmd						: OrderToteCommand;
	
	ton1					: TON;

	ton_heart_beat			: TON;
	bReset_ads_heart_beat	: BOOL;
	bTest					: BOOL;
	
	machine_current_status	: E_PMLState;
	workflow1_status		: ToteSubsystemWorkflowStatus := ToteSubsystemWorkflowStatus.UNKNOWN;
	error1_status			: OrderToteErrorStatus := OrderToteErrorStatus.UNKNOWN;
	
	workflow2_status		: ToteSubsystemWorkflowStatus := ToteSubsystemWorkflowStatus.UNKNOWN;
	error2_status			: OrderToteErrorStatus := OrderToteErrorStatus.UNKNOWN;
	
	loading_tote			: ToteData;
	working1_tote			: ToteData;
	working2_tote			: ToteData;
	
	
	bInbound		: BOOL;
	bOutbound		: BOOL;
	bAbortInbound	: BOOL;
	bAbortOutbound	: BOOL;
	bAutostore_exchange	: BOOL;
	inboundToteParams_temp	: InboundToteParams;
	outboundToteParams_temp	: OutboundToteParams;
	abortToreParams_temp	: AbortToteRequestParams;

	autostore_status	AT%Q* : AutostoreStatus;
	A1	: INT;
	A2	: INT;
	iCase_abort	: INT;
END_VAR

